Yaskawa INFORM job: aprem3TRJ2.JBI

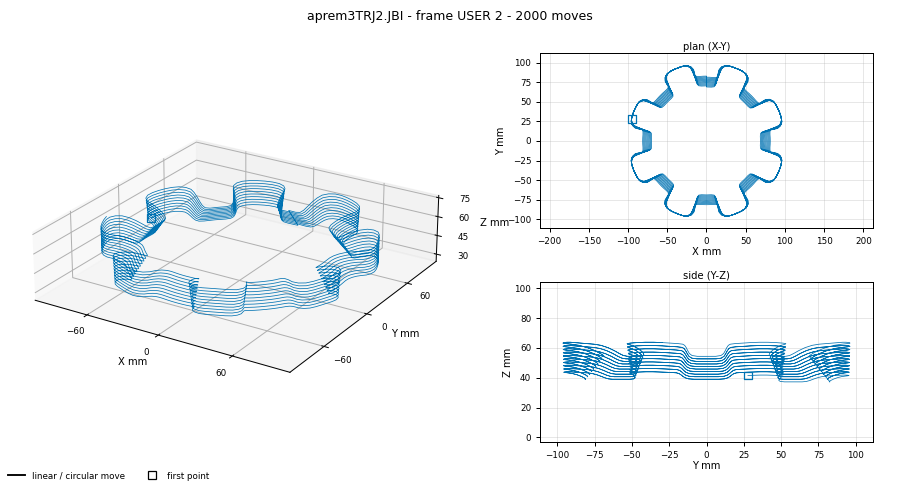
[picture p0: tool path of aprem3TRJ2.JBI in frame USER 2, 2000 of 2000 moves have a stored position in this frame; points joined in program order, loops and branches not executed]
/JOB
//NAME aprem3TRJ2
///FOLDERNAME DEMO
//POS
///NPOS 2000,0,2000,0,0,0
///USER 2
///TOOL 7
///POSTYPE USER
///RECTAN
///RCONF 1,0,0,0,0,0,0,0,0,0,0,0,0,0,0,0,0,0,0,0,0,0,0,0
C00000=-95.500,27.752,41.515,179.9573,-1.4576,-7126.2037
C00001=-94.679,31.992,41.678,179.9802,-0.0621,-7128.6701
C00002=-93.214,36.189,41.785,179.9968,-0.0083,-7131.2180
C00003=-91.502,40.323,41.785,179.9964,-0.0081,-7133.7821
C00004=-89.570,44.326,41.678,179.9701,-0.0579,-7136.3297
C00005=-87.153,47.905,41.515,178.9994,-1.0610,-7138.7961
C00006=-83.964,50.341,41.355,177.9940,-1.0426,-7140.9450
C00007=-80.606,51.270,41.159,176.0647,-0.0633,-7142.4587
C00008=-77.545,50.645,40.789,176.2827,1.1365,-7143.1487
C00009=-74.511,49.565,40.048,179.1830,0.2954,-7143.6320
C00010=-71.724,48.673,39.090,-174.7304,-1.4587,-7144.1614
C00011=-69.261,48.447,38.165,-161.9042,-0.3246,-7144.9722
C00012=-66.868,49.465,37.495,-150.0988,20.4873,-7146.4919
C00013=-64.059,52.288,37.229,-152.5931,29.6910,-7149.2230
C00014=-61.349,55.398,37.217,-152.6199,30.0136,-7152.0820
C00015=-58.451,58.451,37.225,-151.2604,28.7392,-7155.0000
C00016=-55.398,61.349,37.217,-149.9866,27.3805,-7157.9180
C00017=-52.288,64.059,37.229,-150.3100,27.4077,-7160.7770
C00018=-49.465,66.868,37.495,-159.5118,29.9009,-7163.5081
C00019=-48.447,69.261,38.165,179.6754,18.0958,-7165.0278
C00020=-48.673,71.724,39.090,178.5413,5.2696,-7165.8386
C00021=-49.565,74.511,40.048,-179.7046,-0.8170,-7166.3680
C00022=-50.645,77.545,40.789,-178.8635,-3.7173,-7166.8513
C00023=-51.270,80.606,41.159,179.9367,-3.9353,-7167.5413
C00024=-50.341,83.964,41.355,178.9574,-2.0060,-7169.0550
C00025=-47.905,87.153,41.515,178.9390,-1.0006,-7171.2039
C00026=-44.326,89.570,41.678,179.9421,-0.0299,-7173.6703
C00027=-40.323,91.502,41.785,179.9919,-0.0036,-7176.2179
C00028=-36.189,93.214,41.785,179.9917,-0.0032,-7178.7820
C00029=-31.992,94.679,41.678,179.9379,-0.0198,-7181.3299
C00030=-27.752,95.500,41.515,178.5424,-0.0427,-7183.7963
C00031=-23.775,94.968,41.355,177.8447,0.6817,-7185.9450
C00032=-20.743,93.250,41.159,177.1705,2.7402,-7187.4590
C00033=-19.021,90.644,40.789,178.1721,3.4318,-7188.1488
C00034=-17.640,87.735,40.048,179.6311,0.7865,-7188.6317
C00035=-16.299,85.134,39.090,-177.2970,-4.7574,-7189.1618
C00036=-14.718,83.232,38.165,-167.2077,-13.2282,-7189.9720
C00037=-12.305,82.260,37.495,-146.1451,-8.1050,-7191.4924
C00038=-8.324,82.270,37.229,-142.4105,2.0911,-7194.2225
C00039=-4.208,82.553,37.217,-142.2353,2.4190,-7197.0820
C00040=0.000,82.662,37.225,-142.2055,0.0004,-7200.0000
C00041=0.000,81.307,38.958,-141.7581,0.0003,-7200.0000
C00042=4.084,81.202,38.949,-141.7876,-2.4412,-7202.8792
C00043=8.115,80.931,38.962,-141.9747,-1.8578,-7205.7259
C00044=12.050,80.963,39.253,-146.2950,9.3084,-7208.4654
C00045=14.402,82.041,39.987,-169.0753,12.6711,-7209.9566
C00046=15.932,84.113,41.004,-178.0957,3.7141,-7210.7254
C00047=17.234,86.943,42.060,179.2930,-1.6621,-7211.2119
C00048=18.580,90.119,42.880,177.9599,-4.2630,-7211.6495
C00049=20.259,92.987,43.289,176.7690,-3.4884,-7212.2909
C00050=23.317,94.913,43.506,177.4450,-0.9091,-7213.8024
C00051=27.389,95.566,43.684,178.3657,0.0207,-7215.9922
C00052=31.762,94.755,43.864,179.9236,0.0242,-7218.5312
C00053=36.110,93.244,43.984,179.9901,0.0038,-7221.1696
C00054=40.400,91.468,43.984,179.9903,0.0044,-7223.8303
C00055=44.543,89.461,43.864,179.9289,0.0369,-7226.4689
C00056=48.209,86.942,43.684,178.8296,1.1411,-7229.0082
C00057=50.626,83.601,43.506,178.8351,2.4492,-7231.1977
C00058=51.426,80.077,43.289,-179.8173,4.7459,-7232.7089
C00059=50.586,76.861,42.880,-178.4237,4.4542,-7233.3509
C00060=49.291,73.664,42.060,-179.3244,1.6751,-7233.7878
C00061=48.211,70.742,41.004,178.7173,-3.9706,-7234.2746
C00062=47.828,68.195,39.987,178.7113,-16.4605,-7235.0436
C00063=48.729,65.770,39.253,-160.4159,-30.4372,-7236.5348
C00064=51.488,62.965,38.962,-150.0628,-27.9244,-7239.2737
C00065=54.531,60.307,38.949,-149.5942,-27.7685,-7242.1206
C00066=57.493,57.493,38.958,-150.8703,-29.1301,-7245.0000
C00067=60.306,54.531,38.949,-152.2311,-30.4055,-7247.8789
C00068=62.965,51.488,38.962,-152.0747,-29.9361,-7250.7263
C00069=65.770,48.729,39.253,-149.5629,-19.5850,-7253.4652
C00070=68.195,47.828,39.987,-163.5395,1.2887,-7254.9564
C00071=70.742,48.211,41.004,-176.0294,1.2827,-7255.7254
C00072=73.664,49.291,42.060,178.3249,-0.6756,-7256.2122
C00073=76.861,50.586,42.880,175.5458,-1.5763,-7256.6491
C00074=80.077,51.426,43.289,175.2541,-0.1827,-7257.2911
C00075=83.601,50.626,43.506,177.5508,1.1649,-7258.8023
C00076=86.942,48.209,43.684,178.8589,1.1704,-7260.9918
C00077=89.461,44.543,43.864,179.9631,0.0711,-7263.5311
C00078=91.468,40.400,43.984,179.9956,0.0097,-7266.1697
C00079=93.244,36.110,43.984,179.9962,0.0099,-7268.8304
C00080=94.755,31.762,43.864,179.9758,0.0764,-7271.4688
C00081=95.566,27.389,43.684,179.9793,1.6343,-7274.0078
C00082=94.913,23.317,43.506,-179.0909,2.5550,-7276.1976
C00083=92.987,20.259,43.289,-176.5116,3.2310,-7277.7091
C00084=90.119,18.580,42.880,-175.7370,2.0401,-7278.3505
C00085=86.943,17.234,42.060,-178.3379,0.7070,-7278.7881
C00086=84.113,15.932,41.004,176.2859,-1.9043,-7279.2746
C00087=82.041,14.402,39.987,167.3289,-10.9247,-7280.0434
C00088=80.963,12.050,39.253,170.6916,-33.7050,-7281.5346
C00089=80.931,8.115,38.962,-178.1422,-38.0253,-7284.2741
C00090=81.202,4.084,38.949,-177.5588,-38.2124,-7287.1208
C00091=81.307,0.000,38.958,179.9997,-38.2419,-7290.0000
C00092=81.202,-4.084,38.949,177.5593,-38.2124,-7292.8792
C00093=80.931,-8.116,38.962,178.1440,-38.0251,-7295.7266
C00094=80.963,-12.050,39.253,-170.6925,-33.7054,-7298.4654
C00095=82.041,-14.402,39.987,-167.3289,-10.9247,-7299.9566
C00096=84.113,-15.932,41.004,-176.2859,-1.9043,-7300.7254
C00097=86.943,-17.234,42.060,178.3379,0.7070,-7301.2119
C00098=90.119,-18.580,42.880,175.7370,2.0401,-7301.6495
C00099=92.987,-20.259,43.289,176.5116,3.2310,-7302.2909
C00100=94.913,-23.317,43.506,179.0909,2.5550,-7303.8024
C00101=95.566,-27.389,43.684,-179.9793,1.6343,-7305.9922
C00102=94.755,-31.762,43.864,-179.9758,0.0764,-7308.5312
C00103=93.244,-36.110,43.984,-179.9962,0.0099,-7311.1696
C00104=91.468,-40.400,43.984,-179.9956,0.0097,-7313.8303
C00105=89.461,-44.543,43.864,-179.9631,0.0711,-7316.4689
C00106=86.942,-48.209,43.684,-178.8589,1.1704,-7319.0082
C00107=83.601,-50.626,43.506,-177.5508,1.1649,-7321.1977
C00108=80.077,-51.426,43.289,-175.2541,-0.1827,-7322.7089
C00109=76.861,-50.586,42.880,-175.5458,-1.5763,-7323.3509
C00110=73.664,-49.291,42.060,-178.3249,-0.6756,-7323.7878
C00111=70.742,-48.211,41.004,176.0294,1.2827,-7324.2746
C00112=68.195,-47.828,39.987,163.5395,1.2887,-7325.0436
C00113=65.770,-48.729,39.253,149.5628,-19.5841,-7326.5348
C00114=62.965,-51.488,38.962,152.0756,-29.9372,-7329.2737
C00115=60.307,-54.531,38.949,152.2315,-30.4058,-7332.1206
C00116=57.493,-57.493,38.958,150.8699,-29.1297,-7335.0000
C00117=54.531,-60.306,38.949,149.5945,-27.7689,-7337.8789
C00118=51.488,-62.965,38.962,150.0639,-27.9253,-7340.7263
C00119=48.729,-65.770,39.253,160.4150,-30.4371,-7343.4652
C00120=47.828,-68.195,39.987,-178.7113,-16.4605,-7344.9564
C00121=48.211,-70.742,41.004,-178.7173,-3.9706,-7345.7254
C00122=49.291,-73.664,42.060,179.3244,1.6751,-7346.2122
C00123=50.586,-76.861,42.880,178.4237,4.4542,-7346.6491
C00124=51.426,-80.077,43.289,179.8173,4.7459,-7347.2911
C00125=50.626,-83.601,43.506,-178.8351,2.4492,-7348.8023
C00126=48.209,-86.942,43.684,-178.8296,1.1411,-7350.9918
C00127=44.543,-89.461,43.864,-179.9289,0.0369,-7353.5311
C00128=40.400,-91.468,43.984,-179.9903,0.0044,-7356.1697
C00129=36.110,-93.244,43.984,-179.9901,0.0038,-7358.8304
C00130=31.762,-94.755,43.864,-179.9236,0.0242,-7361.4688
C00131=27.389,-95.566,43.684,-178.3657,0.0207,-7364.0078
C00132=23.317,-94.913,43.506,-177.4450,-0.9091,-7366.1976
C00133=20.259,-92.987,43.289,-176.7690,-3.4884,-7367.7091
C00134=18.580,-90.119,42.880,-177.9599,-4.2630,-7368.3505
C00135=17.234,-86.943,42.060,-179.2930,-1.6621,-7368.7881
C00136=15.932,-84.113,41.004,178.0957,3.7141,-7369.2746
C00137=14.402,-82.041,39.987,169.0753,12.6711,-7370.0434
C00138=12.050,-80.963,39.253,146.2950,9.3084,-7371.5346
C00139=8.115,-80.931,38.962,141.9747,-1.8578,-7374.2741
C00140=4.084,-81.202,38.949,141.7876,-2.4412,-7377.1208
C00141=0.000,-81.307,38.958,141.7581,0.0003,-7380.0000
C00142=0.000,-81.307,38.958,141.7581,0.0003,-7380.0000
C00143=-4.084,-81.202,38.949,141.7876,2.4407,-7382.8792
C00144=-8.116,-80.931,38.962,141.9749,1.8560,-7385.7266
C00145=-12.050,-80.963,39.253,146.2946,-9.3075,-7388.4654
C00146=-14.402,-82.041,39.987,169.0753,-12.6711,-7389.9566
C00147=-15.932,-84.113,41.004,178.0957,-3.7141,-7390.7254
C00148=-17.234,-86.943,42.060,-179.2930,1.6621,-7391.2119
C00149=-18.580,-90.119,42.880,-177.9599,4.2630,-7391.6495
C00150=-20.259,-92.987,43.289,-176.7690,3.4884,-7392.2909
C00151=-23.317,-94.913,43.506,-177.4450,0.9091,-7393.8024
C00152=-27.389,-95.566,43.684,-178.3657,-0.0207,-7395.9922
C00153=-31.762,-94.755,43.864,-179.9236,-0.0242,-7398.5312
C00154=-36.110,-93.244,43.984,-179.9901,-0.0038,-7401.1696
C00155=-40.400,-91.468,43.984,-179.9903,-0.0044,-7403.8303
C00156=-44.543,-89.461,43.864,-179.9289,-0.0369,-7406.4689
C00157=-48.209,-86.942,43.684,-178.8296,-1.1411,-7409.0082
C00158=-50.626,-83.601,43.506,-178.8351,-2.4492,-7411.1977
C00159=-51.426,-80.077,43.289,179.8173,-4.7459,-7412.7089
C00160=-50.586,-76.861,42.880,178.4237,-4.4542,-7413.3509
C00161=-49.291,-73.664,42.060,179.3244,-1.6751,-7413.7878
C00162=-48.211,-70.742,41.004,-178.7173,3.9706,-7414.2746
C00163=-47.828,-68.195,39.987,-178.7113,16.4605,-7415.0436
C00164=-48.729,-65.770,39.253,160.4159,30.4372,-7416.5348
C00165=-51.488,-62.965,38.962,150.0628,27.9244,-7419.2737
C00166=-54.531,-60.307,38.949,149.5942,27.7685,-7422.1206
C00167=-57.493,-57.493,38.958,150.8703,29.1301,-7425.0000
C00168=-60.306,-54.531,38.949,152.2311,30.4055,-7427.8789
C00169=-62.965,-51.488,38.962,152.0747,29.9361,-7430.7263
C00170=-65.770,-48.729,39.253,149.5629,19.5850,-7433.4652
C00171=-68.195,-47.828,39.987,163.5395,-1.2887,-7434.9564
C00172=-70.742,-48.211,41.004,176.0294,-1.2827,-7435.7254
C00173=-73.664,-49.291,42.060,-178.3249,0.6756,-7436.2122
C00174=-76.861,-50.586,42.880,-175.5458,1.5763,-7436.6491
C00175=-80.077,-51.426,43.289,-175.2541,0.1827,-7437.2911
C00176=-83.601,-50.626,43.506,-177.5508,-1.1649,-7438.8023
C00177=-86.942,-48.209,43.684,-178.8589,-1.1704,-7440.9918
C00178=-89.461,-44.543,43.864,-179.9631,-0.0711,-7443.5311
C00179=-91.468,-40.400,43.984,-179.9956,-0.0097,-7446.1697
C00180=-93.244,-36.110,43.984,-179.9962,-0.0099,-7448.8304
C00181=-94.755,-31.762,43.864,-179.9758,-0.0764,-7451.4688
C00182=-95.566,-27.389,43.684,-179.9793,-1.6343,-7454.0078
C00183=-94.913,-23.317,43.506,179.0909,-2.5550,-7456.1976
C00184=-92.987,-20.259,43.289,176.5116,-3.2310,-7457.7091
C00185=-90.119,-18.580,42.880,175.7370,-2.0401,-7458.3505
C00186=-86.943,-17.234,42.060,178.3379,-0.7070,-7458.7881
C00187=-84.113,-15.932,41.004,-176.2859,1.9043,-7459.2746
C00188=-82.041,-14.402,39.987,-167.3289,10.9247,-7460.0434
C00189=-80.963,-12.050,39.253,-170.6916,33.7050,-7461.5346
C00190=-80.931,-8.115,38.962,178.1422,38.0253,-7464.2741
C00191=-81.202,-4.084,38.949,177.5588,38.2124,-7467.1208
C00192=-81.307,0.000,38.958,-179.9997,38.2419,-7470.0000
C00193=-81.202,4.084,38.949,-177.5593,38.2124,-7472.8792
C00194=-80.931,8.116,38.962,-178.1440,38.0251,-7475.7266
C00195=-80.963,12.050,39.253,170.6925,33.7054,-7478.4654
C00196=-82.041,14.402,39.987,167.3289,10.9247,-7479.9566
C00197=-84.113,15.932,41.004,176.2859,1.9043,-7480.7254
C00198=-86.943,17.234,42.060,-178.3379,-0.7070,-7481.2119
C00199=-90.119,18.580,42.880,-175.7370,-2.0401,-7481.6495
C00200=-92.987,20.259,43.289,-176.5116,-3.2310,-7482.2909
C00201=-94.913,23.317,43.506,-179.0909,-2.5550,-7483.8024
C00202=-95.566,27.389,43.684,179.9793,-1.6343,-7485.9922
C00203=-94.755,31.762,43.864,179.9758,-0.0764,-7488.5312
C00204=-93.244,36.110,43.984,179.9962,-0.0099,-7491.1696
C00205=-91.468,40.400,43.984,179.9956,-0.0097,-7493.8303
C00206=-89.461,44.543,43.864,179.9631,-0.0711,-7496.4689
C00207=-86.942,48.209,43.684,178.8589,-1.1704,-7499.0082
C00208=-83.601,50.626,43.506,177.5508,-1.1649,-7501.1977
C00209=-80.077,51.426,43.289,175.2541,0.1827,-7502.7089
C00210=-76.861,50.586,42.880,175.5458,1.5763,-7503.3509
C00211=-73.664,49.291,42.060,178.3249,0.6756,-7503.7878
C00212=-70.742,48.211,41.004,-176.0294,-1.2827,-7504.2746
C00213=-68.195,47.828,39.987,-163.5395,-1.2887,-7505.0436
C00214=-65.770,48.729,39.253,-149.5628,19.5841,-7506.5348
C00215=-62.965,51.488,38.962,-152.0756,29.9372,-7509.2737
C00216=-60.307,54.531,38.949,-152.2315,30.4058,-7512.1206
C00217=-57.493,57.493,38.958,-150.8699,29.1297,-7515.0000
C00218=-54.531,60.306,38.949,-149.5945,27.7689,-7517.8789
C00219=-51.488,62.965,38.962,-150.0639,27.9253,-7520.7263
C00220=-48.729,65.770,39.253,-160.4150,30.4371,-7523.4652
C00221=-47.828,68.195,39.987,178.7113,16.4605,-7524.9564
C00222=-48.211,70.742,41.004,178.7173,3.9706,-7525.7254
C00223=-49.291,73.664,42.060,-179.3244,-1.6751,-7526.2122
C00224=-50.586,76.861,42.880,-178.4237,-4.4542,-7526.6491
C00225=-51.426,80.077,43.289,-179.8173,-4.7459,-7527.2911
C00226=-50.626,83.601,43.506,178.8351,-2.4492,-7528.8023
C00227=-48.209,86.942,43.684,178.8296,-1.1411,-7530.9918
C00228=-44.543,89.461,43.864,179.9289,-0.0369,-7533.5311
C00229=-40.400,91.468,43.984,179.9903,-0.0044,-7536.1697
C00230=-36.110,93.244,43.984,179.9901,-0.0038,-7538.8304
C00231=-31.762,94.755,43.864,179.9236,-0.0242,-7541.4688
C00232=-27.389,95.566,43.684,178.3657,-0.0207,-7544.0078
C00233=-23.317,94.913,43.506,177.4450,0.9091,-7546.1976
C00234=-20.259,92.987,43.289,176.7690,3.4884,-7547.7091
C00235=-18.580,90.119,42.880,177.9599,4.2630,-7548.3505
C00236=-17.234,86.943,42.060,179.2930,1.6621,-7548.7881
C00237=-15.932,84.113,41.004,-178.0957,-3.7141,-7549.2746
C00238=-14.402,82.041,39.987,-169.0753,-12.6711,-7550.0434
C00239=-12.050,80.963,39.253,-146.2946,-9.3075,-7551.5346
C00240=-8.116,80.931,38.962,-141.9749,1.8560,-7554.2734
C00241=-4.084,81.202,38.949,-141.7876,2.4407,-7557.1208
C00242=0.000,81.307,38.958,-141.7581,0.0003,-7560.0000
C00243=0.000,79.940,40.681,-141.3945,0.0003,-7560.0000
C00244=3.959,79.840,40.672,-141.4236,-2.4543,-7562.8388
C00245=7.905,79.580,40.686,-141.6255,-1.5989,-7565.6728
C00246=11.791,79.654,41.003,-146.5959,10.4668,-7568.4202
C00247=14.083,80.839,41.802,-170.8088,11.8957,-7569.8823
C00248=15.561,83.082,42.912,-178.7432,2.6994,-7570.6084
C00249=16.825,86.143,44.068,179.0449,-2.4598,-7571.0516
C00250=18.134,89.588,44.968,177.8329,-5.0059,-7571.4429
C00251=19.771,92.721,45.418,176.4774,-4.2024,-7572.0370
C00252=22.856,94.857,45.657,177.0847,-1.1491,-7573.5473
C00253=27.022,95.633,45.852,178.2015,-0.0057,-7575.7781
C00254=31.529,94.831,46.051,179.9101,0.0282,-7578.3907
C00255=36.031,93.275,46.182,179.9885,0.0043,-7581.1209
C00256=40.478,91.433,46.182,179.9888,0.0050,-7583.8793
C00257=44.762,89.350,46.051,179.9165,0.0436,-7586.6097
C00258=48.515,86.730,45.852,178.7321,1.2760,-7589.2218
C00259=50.913,83.236,45.657,178.7496,2.8735,-7591.4529
C00260=51.583,79.544,45.418,-179.5172,5.4544,-7592.9628
C00261=50.526,76.172,44.968,-177.9852,5.0686,-7593.5569
C00262=49.015,72.810,44.068,-178.9351,2.4144,-7593.9481
C00263=47.744,69.752,42.912,178.9787,-2.7968,-7594.3909
C00264=47.203,67.120,41.802,178.0217,-14.7549,-7595.1173
C00265=47.986,64.662,41.003,-161.4435,-30.8352,-7596.5793
C00266=50.682,61.862,40.686,-149.9004,-28.3778,-7599.3269
C00267=53.655,59.255,40.672,-149.2767,-28.0885,-7602.1606
C00268=56.526,56.526,40.681,-150.5516,-29.4487,-7605.0000
C00269=59.255,53.656,40.672,-151.9113,-30.7231,-7607.8388
C00270=61.862,50.682,40.686,-151.6213,-30.0984,-7610.6731
C00271=64.662,47.986,41.003,-149.1649,-18.5575,-7613.4207
C00272=67.120,47.203,41.802,-165.2451,1.9783,-7614.8827
C00273=69.752,47.744,42.912,-177.2032,1.0213,-7615.6091
C00274=72.810,49.015,44.068,177.5856,-1.0649,-7616.0519
C00275=76.172,50.526,44.968,174.9314,-2.0148,-7616.4431
C00276=79.544,51.583,45.418,174.5456,-0.4828,-7617.0372
C00277=83.236,50.913,45.657,177.1265,1.2504,-7618.5471
C00278=86.730,48.515,45.852,178.7240,1.2679,-7620.7782
C00279=89.350,44.762,46.051,179.9564,0.0835,-7623.3903
C00280=91.433,40.478,46.182,179.9950,0.0112,-7626.1207
C00281=93.275,36.031,46.182,179.9957,0.0115,-7628.8791
C00282=94.831,31.529,46.051,179.9718,0.0899,-7631.6093
C00283=95.633,27.022,45.852,-179.9943,1.7985,-7634.2219
C00284=94.857,22.856,45.657,-178.8509,2.9153,-7636.4527
C00285=92.721,19.771,45.418,-175.7976,3.5226,-7637.9630
C00286=89.588,18.134,44.968,-174.9941,2.1671,-7638.5571
C00287=86.143,16.825,44.068,-177.5402,0.9551,-7638.9484
C00288=83.082,15.561,42.912,177.3006,-1.2568,-7639.3916
C00289=80.839,14.083,41.802,168.1043,-9.1912,-7640.1177
C00290=79.654,11.791,41.003,169.5332,-33.4041,-7641.5798
C00291=79.580,7.905,40.686,-178.4011,-38.3745,-7644.3272
C00292=79.840,3.959,40.672,-177.5457,-38.5764,-7647.1612
C00293=79.940,0.000,40.681,179.9997,-38.6055,-7650.0000
C00294=79.840,-3.959,40.672,177.5462,-38.5764,-7652.8388
C00295=79.580,-7.905,40.686,178.4031,-38.3743,-7655.6728
C00296=79.654,-11.792,41.003,-169.5340,-33.4045,-7658.4209
C00297=80.839,-14.083,41.802,-168.1043,-9.1912,-7659.8823
C00298=83.082,-15.561,42.912,-177.3006,-1.2568,-7660.6084
C00299=86.143,-16.825,44.068,177.5402,0.9551,-7661.0516
C00300=89.588,-18.134,44.968,174.9941,2.1671,-7661.4429
C00301=92.721,-19.771,45.418,175.7976,3.5226,-7662.0370
C00302=94.857,-22.856,45.657,178.8509,2.9153,-7663.5473
C00303=95.633,-27.022,45.852,179.9943,1.7985,-7665.7781
C00304=94.831,-31.529,46.051,-179.9718,0.0899,-7668.3907
C00305=93.275,-36.031,46.182,-179.9957,0.0115,-7671.1209
C00306=91.433,-40.478,46.182,-179.9950,0.0112,-7673.8793
C00307=89.350,-44.762,46.051,-179.9564,0.0835,-7676.6097
C00308=86.730,-48.515,45.852,-178.7240,1.2679,-7679.2218
C00309=83.236,-50.913,45.657,-177.1265,1.2504,-7681.4529
C00310=79.544,-51.583,45.418,-174.5456,-0.4828,-7682.9628
C00311=76.172,-50.526,44.968,-174.9314,-2.0148,-7683.5569
C00312=72.810,-49.015,44.068,-177.5856,-1.0649,-7683.9481
C00313=69.752,-47.744,42.912,177.2032,1.0213,-7684.3909
C00314=67.120,-47.203,41.802,165.2451,1.9783,-7685.1173
C00315=64.662,-47.986,41.003,149.1648,-18.5565,-7686.5793
C00316=61.862,-50.682,40.686,151.6222,-30.0996,-7689.3269
C00317=59.255,-53.655,40.672,151.9115,-30.7233,-7692.1606
C00318=56.526,-56.526,40.681,150.5513,-29.4484,-7695.0000
C00319=53.656,-59.255,40.672,149.2769,-28.0887,-7697.8388
C00320=50.682,-61.862,40.686,149.9016,-28.3787,-7700.6731
C00321=47.986,-64.662,41.003,161.4425,-30.8351,-7703.4207
C00322=47.203,-67.120,41.802,-178.0217,-14.7549,-7704.8827
C00323=47.744,-69.752,42.912,-178.9787,-2.7968,-7705.6091
C00324=49.015,-72.810,44.068,178.9351,2.4144,-7706.0519
C00325=50.526,-76.172,44.968,177.9852,5.0686,-7706.4431
C00326=51.583,-79.544,45.418,179.5172,5.4544,-7707.0372
C00327=50.913,-83.236,45.657,-178.7496,2.8735,-7708.5471
C00328=48.515,-86.730,45.852,-178.7321,1.2760,-7710.7782
C00329=44.762,-89.350,46.051,-179.9165,0.0436,-7713.3903
C00330=40.478,-91.433,46.182,-179.9888,0.0050,-7716.1207
C00331=36.031,-93.275,46.182,-179.9885,0.0043,-7718.8791
C00332=31.529,-94.831,46.051,-179.9101,0.0282,-7721.6093
C00333=27.022,-95.633,45.852,-178.2015,-0.0057,-7724.2219
C00334=22.856,-94.857,45.657,-177.0847,-1.1491,-7726.4527
C00335=19.771,-92.721,45.418,-176.4774,-4.2024,-7727.9630
C00336=18.134,-89.588,44.968,-177.8329,-5.0059,-7728.5571
C00337=16.825,-86.143,44.068,-179.0449,-2.4598,-7728.9484
C00338=15.561,-83.082,42.912,178.7432,2.6994,-7729.3916
C00339=14.083,-80.839,41.802,170.8088,11.8957,-7730.1177
C00340=11.791,-79.654,41.003,146.5959,10.4668,-7731.5798
C00341=7.905,-79.580,40.686,141.6255,-1.5989,-7734.3272
C00342=3.959,-79.840,40.672,141.4236,-2.4543,-7737.1612
C00343=0.000,-79.940,40.681,141.3945,0.0003,-7740.0000
C00344=0.000,-79.940,40.681,141.3945,0.0003,-7740.0000
C00345=-3.959,-79.840,40.672,141.4236,2.4538,-7742.8388
C00346=-7.905,-79.580,40.686,141.6257,1.5969,-7745.6728
C00347=-11.792,-79.654,41.003,146.5955,-10.4660,-7748.4209
C00348=-14.083,-80.839,41.802,170.8088,-11.8957,-7749.8823
C00349=-15.561,-83.082,42.912,178.7432,-2.6994,-7750.6084
C00350=-16.825,-86.143,44.068,-179.0449,2.4598,-7751.0516
C00351=-18.134,-89.588,44.968,-177.8329,5.0059,-7751.4429
C00352=-19.771,-92.721,45.418,-176.4774,4.2024,-7752.0370
C00353=-22.856,-94.857,45.657,-177.0847,1.1491,-7753.5473
C00354=-27.022,-95.633,45.852,-178.2015,0.0057,-7755.7781
C00355=-31.529,-94.831,46.051,-179.9101,-0.0282,-7758.3907
C00356=-36.031,-93.275,46.182,-179.9885,-0.0043,-7761.1209
C00357=-40.478,-91.433,46.182,-179.9888,-0.0050,-7763.8793
C00358=-44.762,-89.350,46.051,-179.9165,-0.0436,-7766.6097
C00359=-48.515,-86.730,45.852,-178.7321,-1.2760,-7769.2218
C00360=-50.913,-83.236,45.657,-178.7496,-2.8735,-7771.4529
C00361=-51.583,-79.544,45.418,179.5172,-5.4544,-7772.9628
C00362=-50.526,-76.172,44.968,177.9852,-5.0686,-7773.5569
C00363=-49.015,-72.810,44.068,178.9351,-2.4144,-7773.9481
C00364=-47.744,-69.752,42.912,-178.9787,2.7968,-7774.3909
C00365=-47.203,-67.120,41.802,-178.0217,14.7549,-7775.1173
C00366=-47.986,-64.662,41.003,161.4435,30.8352,-7776.5793
C00367=-50.682,-61.862,40.686,149.9004,28.3778,-7779.3269
C00368=-53.655,-59.255,40.672,149.2767,28.0885,-7782.1606
C00369=-56.526,-56.526,40.681,150.5516,29.4487,-7785.0000
C00370=-59.255,-53.656,40.672,151.9113,30.7231,-7787.8388
C00371=-61.862,-50.682,40.686,151.6213,30.0984,-7790.6731
C00372=-64.662,-47.986,41.003,149.1649,18.5575,-7793.4207
C00373=-67.120,-47.203,41.802,165.2451,-1.9783,-7794.8827
C00374=-69.752,-47.744,42.912,177.2032,-1.0213,-7795.6091
C00375=-72.810,-49.015,44.068,-177.5856,1.0649,-7796.0519
C00376=-76.172,-50.526,44.968,-174.9314,2.0148,-7796.4431
C00377=-79.544,-51.583,45.418,-174.5456,0.4828,-7797.0372
C00378=-83.236,-50.913,45.657,-177.1265,-1.2504,-7798.5471
C00379=-86.730,-48.515,45.852,-178.7240,-1.2679,-7800.7782
C00380=-89.350,-44.762,46.051,-179.9564,-0.0835,-7803.3903
C00381=-91.433,-40.478,46.182,-179.9950,-0.0112,-7806.1207
C00382=-93.275,-36.031,46.182,-179.9957,-0.0115,-7808.8791
C00383=-94.831,-31.529,46.051,-179.9718,-0.0899,-7811.6093
C00384=-95.633,-27.022,45.852,179.9943,-1.7985,-7814.2219
C00385=-94.857,-22.856,45.657,178.8509,-2.9153,-7816.4527
C00386=-92.721,-19.771,45.418,175.7976,-3.5226,-7817.9630
C00387=-89.588,-18.134,44.968,174.9941,-2.1671,-7818.5571
C00388=-86.143,-16.825,44.068,177.5402,-0.9551,-7818.9484
C00389=-83.082,-15.561,42.912,-177.3006,1.2568,-7819.3916
C00390=-80.839,-14.083,41.802,-168.1043,9.1912,-7820.1177
C00391=-79.654,-11.791,41.003,-169.5332,33.4041,-7821.5798
C00392=-79.580,-7.905,40.686,178.4011,38.3745,-7824.3272
C00393=-79.840,-3.959,40.672,177.5457,38.5764,-7827.1612
C00394=-79.940,0.000,40.681,-179.9997,38.6055,-7830.0000
C00395=-79.840,3.959,40.672,-177.5462,38.5764,-7832.8388
C00396=-79.580,7.905,40.686,-178.4031,38.3743,-7835.6728
C00397=-79.654,11.792,41.003,169.5340,33.4045,-7838.4209
C00398=-80.839,14.083,41.802,168.1043,9.1912,-7839.8823
C00399=-83.082,15.561,42.912,177.3006,1.2568,-7840.6084
C00400=-86.143,16.825,44.068,-177.5402,-0.9551,-7841.0516
C00401=-89.588,18.134,44.968,-174.9941,-2.1671,-7841.4429
C00402=-92.721,19.771,45.418,-175.7976,-3.5226,-7842.0370
C00403=-94.857,22.856,45.657,-178.8509,-2.9153,-7843.5473
C00404=-95.633,27.022,45.852,-179.9943,-1.7985,-7845.7781
C00405=-94.831,31.529,46.051,179.9718,-0.0899,-7848.3907
C00406=-93.275,36.031,46.182,179.9957,-0.0115,-7851.1209
C00407=-91.433,40.478,46.182,179.9950,-0.0112,-7853.8793
C00408=-89.350,44.762,46.051,179.9564,-0.0835,-7856.6097
C00409=-86.730,48.515,45.852,178.7240,-1.2679,-7859.2218
C00410=-83.236,50.913,45.657,177.1265,-1.2504,-7861.4529
C00411=-79.544,51.583,45.418,174.5456,0.4828,-7862.9628
C00412=-76.172,50.526,44.968,174.9314,2.0148,-7863.5569
C00413=-72.810,49.015,44.068,177.5856,1.0649,-7863.9481
C00414=-69.752,47.744,42.912,-177.2032,-1.0213,-7864.3909
C00415=-67.120,47.203,41.802,-165.2451,-1.9783,-7865.1173
C00416=-64.662,47.986,41.003,-149.1648,18.5565,-7866.5793
C00417=-61.862,50.682,40.686,-151.6222,30.0996,-7869.3269
C00418=-59.255,53.655,40.672,-151.9115,30.7233,-7872.1606
C00419=-56.526,56.526,40.681,-150.5513,29.4484,-7875.0000
C00420=-53.656,59.255,40.672,-149.2769,28.0887,-7877.8388
C00421=-50.682,61.862,40.686,-149.9016,28.3787,-7880.6731
C00422=-47.986,64.662,41.003,-161.4425,30.8351,-7883.4207
C00423=-47.203,67.120,41.802,178.0217,14.7549,-7884.8827
C00424=-47.744,69.752,42.912,178.9787,2.7968,-7885.6091
C00425=-49.015,72.810,44.068,-178.9351,-2.4144,-7886.0519
C00426=-50.526,76.172,44.968,-177.9852,-5.0686,-7886.4431
C00427=-51.583,79.544,45.418,-179.5172,-5.4544,-7887.0372
C00428=-50.913,83.236,45.657,178.7496,-2.8735,-7888.5471
C00429=-48.515,86.730,45.852,178.7321,-1.2760,-7890.7782
C00430=-44.762,89.350,46.051,179.9165,-0.0436,-7893.3903
C00431=-40.478,91.433,46.182,179.9888,-0.0050,-7896.1207
C00432=-36.031,93.275,46.182,179.9885,-0.0043,-7898.8791
C00433=-31.529,94.831,46.051,179.9101,-0.0282,-7901.6093
C00434=-27.022,95.633,45.852,178.2015,0.0057,-7904.2219
C00435=-22.856,94.857,45.657,177.0847,1.1491,-7906.4527
C00436=-19.771,92.721,45.418,176.4774,4.2024,-7907.9630
C00437=-18.134,89.588,44.968,177.8329,5.0059,-7908.5571
C00438=-16.825,86.143,44.068,179.0449,2.4598,-7908.9484
C00439=-15.561,83.082,42.912,-178.7432,-2.6994,-7909.3916
C00440=-14.083,80.839,41.802,-170.8088,-11.8957,-7910.1177
C00441=-11.792,79.654,41.003,-146.5955,-10.4660,-7911.5791
C00442=-7.905,79.580,40.686,-141.6257,1.5969,-7914.3272
C00443=-3.959,79.840,40.672,-141.4236,2.4538,-7917.1612
C00444=0.000,79.940,40.681,-141.3945,0.0003,-7920.0000
C00445=0.000,78.562,42.397,-141.1109,0.0002,-7920.0000
C00446=3.833,78.467,42.387,-141.1396,-2.4588,-7922.7966
C00447=7.694,78.220,42.402,-141.3590,-1.3181,-7925.6177
C00448=11.532,78.336,42.745,-147.0431,11.5605,-7928.3745
C00449=13.762,79.628,43.611,-172.3770,10.9592,-7929.8055
C00450=15.189,82.045,44.816,-179.2626,1.7346,-7930.4884
C00451=16.414,85.339,46.074,178.8680,-3.1755,-7930.8872
C00452=17.687,89.056,47.055,177.7717,-5.6565,-7931.2331
C00453=19.281,92.454,47.546,176.2826,-4.8619,-7931.7800
C00454=22.392,94.802,47.807,176.7679,-1.3940,-7933.2896
C00455=26.654,95.700,48.020,178.0518,-0.0356,-7935.5634
C00456=31.296,94.909,48.237,179.8977,0.0319,-7938.2498
C00457=35.952,93.306,48.381,179.9872,0.0049,-7941.0723
C00458=40.555,91.399,48.381,179.9875,0.0056,-7943.9275
C00459=44.981,89.240,48.237,179.9051,0.0498,-7946.7502
C00460=48.823,86.517,48.020,178.6473,1.4030,-7949.4368
C00461=51.201,82.869,47.807,178.6983,3.2702,-7951.7100
C00462=51.741,79.009,47.546,-179.1862,6.0558,-7953.2198
C00463=50.465,75.478,47.055,-177.5651,5.5716,-7953.7669
C00464=48.737,71.950,46.074,-178.5531,3.0453,-7954.1127
C00465=47.275,68.755,44.816,179.2946,-1.7479,-7954.5119
C00466=46.575,66.037,43.611,177.5785,-13.0378,-7955.1948
C00467=47.238,63.546,42.745,-162.5779,-31.0935,-7956.6259
C00468=49.870,60.750,42.402,-149.8188,-28.7683,-7959.3828
C00469=52.774,58.195,42.387,-149.0312,-28.3421,-7962.2032
C00470=55.552,55.552,42.397,-150.3022,-29.6980,-7965.0000
C00471=58.195,52.774,42.387,-151.6576,-30.9686,-7967.7968
C00472=60.750,49.870,42.402,-151.2308,-30.1799,-7970.6172
C00473=63.546,47.238,42.745,-148.9065,-17.4230,-7973.3741
C00474=66.037,46.575,43.611,-166.9622,2.4215,-7974.8052
C00475=68.755,47.275,44.816,-178.2521,0.7054,-7975.4881
C00476=71.950,48.737,46.074,176.9547,-1.4469,-7975.8873
C00477=75.478,50.465,47.055,174.4284,-2.4349,-7976.2331
C00478=79.009,51.741,47.546,173.9442,-0.8138,-7976.7802
C00479=82.869,51.201,47.807,176.7298,1.3017,-7978.2900
C00480=86.517,48.823,48.020,178.5970,1.3527,-7980.5632
C00481=89.240,44.981,48.237,179.9502,0.0949,-7983.2498
C00482=91.399,40.555,48.381,179.9944,0.0125,-7986.0725
C00483=93.306,35.952,48.381,179.9951,0.0128,-7988.9277
C00484=94.909,31.296,48.237,179.9681,0.1023,-7991.7502
C00485=95.700,26.654,48.020,-179.9644,1.9482,-7994.4366
C00486=94.802,22.392,47.807,-178.6060,3.2321,-7996.7104
C00487=92.454,19.281,47.546,-175.1381,3.7174,-7998.2200
C00488=89.056,17.687,47.055,-174.3435,2.2283,-7998.7669
C00489=85.339,16.414,46.074,-176.8245,1.1320,-7999.1128
C00490=82.045,15.189,44.816,178.2654,-0.7374,-7999.5116
C00491=79.628,13.762,43.611,169.0408,-7.6230,-8000.1945
C00492=78.336,11.532,42.745,168.4395,-32.9569,-8001.6255
C00493=78.220,7.694,42.402,-178.6819,-38.6410,-8004.3823
C00494=78.467,3.833,42.387,-177.5412,-38.8604,-8007.2034
C00495=78.562,0.000,42.397,179.9998,-38.8891,-8010.0000
C00496=78.467,-3.833,42.387,177.5416,-38.8604,-8012.7966
C00497=78.220,-7.694,42.402,178.6839,-38.6407,-8015.6177
C00498=78.336,-11.532,42.745,-168.4403,-32.9573,-8018.3745
C00499=79.628,-13.762,43.611,-169.0408,-7.6230,-8019.8055
C00500=82.045,-15.189,44.816,-178.2654,-0.7374,-8020.4884
C00501=85.339,-16.414,46.074,176.8245,1.1320,-8020.8872
C00502=89.056,-17.687,47.055,174.3435,2.2283,-8021.2331
C00503=92.454,-19.281,47.546,175.1381,3.7174,-8021.7800
C00504=94.802,-22.392,47.807,178.6060,3.2321,-8023.2896
C00505=95.700,-26.654,48.020,179.9644,1.9482,-8025.5634
C00506=94.909,-31.296,48.237,-179.9681,0.1023,-8028.2498
C00507=93.306,-35.952,48.381,-179.9951,0.0128,-8031.0723
C00508=91.399,-40.555,48.381,-179.9944,0.0125,-8033.9275
C00509=89.240,-44.981,48.237,-179.9502,0.0949,-8036.7502
C00510=86.517,-48.823,48.020,-178.5970,1.3527,-8039.4368
C00511=82.869,-51.201,47.807,-176.7298,1.3017,-8041.7100
C00512=79.009,-51.741,47.546,-173.9442,-0.8138,-8043.2198
C00513=75.478,-50.465,47.055,-174.4284,-2.4349,-8043.7669
C00514=71.950,-48.737,46.074,-176.9547,-1.4469,-8044.1127
C00515=68.755,-47.275,44.816,178.2521,0.7054,-8044.5119
C00516=66.037,-46.575,43.611,166.9622,2.4215,-8045.1948
C00517=63.546,-47.238,42.745,148.9065,-17.4221,-8046.6259
C00518=60.750,-49.870,42.402,151.2317,-30.1812,-8049.3828
C00519=58.195,-52.774,42.387,151.6579,-30.9688,-8052.2032
C00520=55.552,-55.552,42.397,150.3020,-29.6978,-8055.0000
C00521=52.774,-58.195,42.387,149.0314,-28.3424,-8057.7968
C00522=49.870,-60.750,42.402,149.8201,-28.7692,-8060.6172
C00523=47.238,-63.546,42.745,162.5770,-31.0935,-8063.3741
C00524=46.575,-66.037,43.611,-177.5785,-13.0378,-8064.8052
C00525=47.275,-68.755,44.816,-179.2946,-1.7479,-8065.4881
C00526=48.737,-71.950,46.074,178.5531,3.0453,-8065.8873
C00527=50.465,-75.478,47.055,177.5651,5.5716,-8066.2331
C00528=51.741,-79.009,47.546,179.1862,6.0558,-8066.7802
C00529=51.201,-82.869,47.807,-178.6983,3.2702,-8068.2900
C00530=48.823,-86.517,48.020,-178.6473,1.4030,-8070.5632
C00531=44.981,-89.240,48.237,-179.9051,0.0498,-8073.2498
C00532=40.555,-91.399,48.381,-179.9875,0.0056,-8076.0725
C00533=35.952,-93.306,48.381,-179.9872,0.0049,-8078.9277
C00534=31.296,-94.909,48.237,-179.8977,0.0319,-8081.7502
C00535=26.654,-95.700,48.020,-178.0518,-0.0356,-8084.4366
C00536=22.392,-94.802,47.807,-176.7679,-1.3940,-8086.7104
C00537=19.281,-92.454,47.546,-176.2826,-4.8619,-8088.2200
C00538=17.687,-89.056,47.055,-177.7717,-5.6565,-8088.7669
C00539=16.414,-85.339,46.074,-178.8680,-3.1755,-8089.1128
C00540=15.189,-82.045,44.816,179.2626,1.7346,-8089.5116
C00541=13.762,-79.628,43.611,172.3770,10.9592,-8090.1945
C00542=11.532,-78.336,42.745,147.0431,11.5605,-8091.6255
C00543=7.694,-78.220,42.402,141.3590,-1.3181,-8094.3823
C00544=3.833,-78.467,42.387,141.1396,-2.4588,-8097.2034
C00545=0.000,-78.562,42.397,141.1109,0.0002,-8100.0000
C00546=0.000,-78.562,42.397,141.1109,0.0002,-8100.0000
C00547=-3.833,-78.467,42.387,141.1396,2.4584,-8102.7966
C00548=-7.694,-78.220,42.402,141.3593,1.3161,-8105.6177
C00549=-11.532,-78.336,42.745,147.0427,-11.5597,-8108.3745
C00550=-13.762,-79.628,43.611,172.3770,-10.9592,-8109.8055
C00551=-15.189,-82.045,44.816,179.2626,-1.7346,-8110.4884
C00552=-16.414,-85.339,46.074,-178.8680,3.1755,-8110.8872
C00553=-17.687,-89.056,47.055,-177.7717,5.6565,-8111.2331
C00554=-19.281,-92.454,47.546,-176.2826,4.8619,-8111.7800
C00555=-22.392,-94.802,47.807,-176.7679,1.3940,-8113.2896
C00556=-26.654,-95.700,48.020,-178.0518,0.0356,-8115.5634
C00557=-31.296,-94.909,48.237,-179.8977,-0.0319,-8118.2498
C00558=-35.952,-93.306,48.381,-179.9872,-0.0049,-8121.0723
C00559=-40.555,-91.399,48.381,-179.9875,-0.0056,-8123.9275
C00560=-44.981,-89.240,48.237,-179.9051,-0.0498,-8126.7502
C00561=-48.823,-86.517,48.020,-178.6473,-1.4030,-8129.4368
C00562=-51.201,-82.869,47.807,-178.6983,-3.2702,-8131.7100
C00563=-51.741,-79.009,47.546,179.1862,-6.0558,-8133.2198
C00564=-50.465,-75.478,47.055,177.5651,-5.5716,-8133.7669
C00565=-48.737,-71.950,46.074,178.5531,-3.0453,-8134.1127
C00566=-47.275,-68.755,44.816,-179.2946,1.7479,-8134.5119
C00567=-46.575,-66.037,43.611,-177.5785,13.0378,-8135.1948
C00568=-47.238,-63.546,42.745,162.5779,31.0935,-8136.6259
C00569=-49.870,-60.750,42.402,149.8188,28.7683,-8139.3828
C00570=-52.774,-58.195,42.387,149.0312,28.3421,-8142.2032
C00571=-55.552,-55.552,42.397,150.3022,29.6980,-8145.0000
C00572=-58.195,-52.774,42.387,151.6576,30.9686,-8147.7968
C00573=-60.750,-49.870,42.402,151.2308,30.1799,-8150.6172
C00574=-63.546,-47.238,42.745,148.9065,17.4230,-8153.3741
C00575=-66.037,-46.575,43.611,166.9622,-2.4215,-8154.8052
C00576=-68.755,-47.275,44.816,178.2521,-0.7054,-8155.4881
C00577=-71.950,-48.737,46.074,-176.9547,1.4469,-8155.8873
C00578=-75.478,-50.465,47.055,-174.4284,2.4349,-8156.2331
C00579=-79.009,-51.741,47.546,-173.9442,0.8138,-8156.7802
C00580=-82.869,-51.201,47.807,-176.7298,-1.3017,-8158.2900
C00581=-86.517,-48.823,48.020,-178.5970,-1.3527,-8160.5632
C00582=-89.240,-44.981,48.237,-179.9502,-0.0949,-8163.2498
C00583=-91.399,-40.555,48.381,-179.9944,-0.0125,-8166.0725
C00584=-93.306,-35.952,48.381,-179.9951,-0.0128,-8168.9277
C00585=-94.909,-31.296,48.237,-179.9681,-0.1023,-8171.7502
C00586=-95.700,-26.654,48.020,179.9644,-1.9482,-8174.4366
C00587=-94.802,-22.392,47.807,178.6060,-3.2321,-8176.7104
C00588=-92.454,-19.281,47.546,175.1381,-3.7174,-8178.2200
C00589=-89.056,-17.687,47.055,174.3435,-2.2283,-8178.7669
C00590=-85.339,-16.414,46.074,176.8245,-1.1320,-8179.1128
C00591=-82.045,-15.189,44.816,-178.2654,0.7374,-8179.5116
C00592=-79.628,-13.762,43.611,-169.0408,7.6230,-8180.1945
C00593=-78.336,-11.532,42.745,-168.4395,32.9569,-8181.6255
C00594=-78.220,-7.694,42.402,178.6819,38.6410,-8184.3823
C00595=-78.467,-3.833,42.387,177.5412,38.8604,-8187.2034
C00596=-78.562,0.000,42.397,-179.9998,38.8891,-8190.0000
C00597=-78.467,3.833,42.387,-177.5416,38.8604,-8192.7966
C00598=-78.220,7.694,42.402,-178.6839,38.6407,-8195.6177
C00599=-78.336,11.532,42.745,168.4403,32.9573,-8198.3745
C00600=-79.628,13.762,43.611,169.0408,7.6230,-8199.8055
C00601=-82.045,15.189,44.816,178.2654,0.7374,-8200.4884
C00602=-85.339,16.414,46.074,-176.8245,-1.1320,-8200.8872
C00603=-89.056,17.687,47.055,-174.3435,-2.2283,-8201.2331
C00604=-92.454,19.281,47.546,-175.1381,-3.7174,-8201.7800
C00605=-94.802,22.392,47.807,-178.6060,-3.2321,-8203.2896
C00606=-95.700,26.654,48.020,-179.9644,-1.9482,-8205.5634
C00607=-94.909,31.296,48.237,179.9681,-0.1023,-8208.2498
C00608=-93.306,35.952,48.381,179.9951,-0.0128,-8211.0723
C00609=-91.399,40.555,48.381,179.9944,-0.0125,-8213.9275
C00610=-89.240,44.981,48.237,179.9502,-0.0949,-8216.7502
C00611=-86.517,48.823,48.020,178.5970,-1.3527,-8219.4368
C00612=-82.869,51.201,47.807,176.7298,-1.3017,-8221.7100
C00613=-79.009,51.741,47.546,173.9442,0.8138,-8223.2198
C00614=-75.478,50.465,47.055,174.4284,2.4349,-8223.7669
C00615=-71.950,48.737,46.074,176.9547,1.4469,-8224.1127
C00616=-68.755,47.275,44.816,-178.2521,-0.7054,-8224.5119
C00617=-66.037,46.575,43.611,-166.9622,-2.4215,-8225.1948
C00618=-63.546,47.238,42.745,-148.9065,17.4221,-8226.6259
C00619=-60.750,49.870,42.402,-151.2317,30.1812,-8229.3828
C00620=-58.195,52.774,42.387,-151.6579,30.9688,-8232.2032
C00621=-55.552,55.552,42.397,-150.3020,29.6978,-8235.0000
C00622=-52.774,58.195,42.387,-149.0314,28.3424,-8237.7968
C00623=-49.870,60.750,42.402,-149.8201,28.7692,-8240.6172
C00624=-47.238,63.546,42.745,-162.5770,31.0935,-8243.3741
C00625=-46.575,66.037,43.611,177.5785,13.0378,-8244.8052
C00626=-47.275,68.755,44.816,179.2946,1.7479,-8245.4881
C00627=-48.737,71.950,46.074,-178.5531,-3.0453,-8245.8873
C00628=-50.465,75.478,47.055,-177.5651,-5.5716,-8246.2331
C00629=-51.741,79.009,47.546,-179.1862,-6.0558,-8246.7802
C00630=-51.201,82.869,47.807,178.6983,-3.2702,-8248.2900
C00631=-48.823,86.517,48.020,178.6473,-1.4030,-8250.5632
C00632=-44.981,89.240,48.237,179.9051,-0.0498,-8253.2498
C00633=-40.555,91.399,48.381,179.9875,-0.0056,-8256.0725
C00634=-35.952,93.306,48.381,179.9872,-0.0049,-8258.9277
C00635=-31.296,94.909,48.237,179.8977,-0.0319,-8261.7502
C00636=-26.654,95.700,48.020,178.0518,0.0356,-8264.4366
C00637=-22.392,94.802,47.807,176.7679,1.3940,-8266.7104
C00638=-19.281,92.454,47.546,176.2826,4.8619,-8268.2200
C00639=-17.687,89.056,47.055,177.7717,5.6565,-8268.7669
C00640=-16.414,85.339,46.074,178.8680,3.1755,-8269.1128
C00641=-15.189,82.045,44.816,-179.2626,-1.7346,-8269.5116
C00642=-13.762,79.628,43.611,-172.3770,-10.9592,-8270.1945
C00643=-11.532,78.336,42.745,-147.0427,-11.5597,-8271.6255
C00644=-7.694,78.220,42.402,-141.3593,1.3161,-8274.3823
C00645=-3.833,78.467,42.387,-141.1396,2.4584,-8277.2034
C00646=0.000,78.562,42.397,-141.1109,0.0002,-8280.0000
C00647=0.000,77.178,44.107,-140.9045,0.0002,-8280.0000
C00648=3.707,77.088,44.096,-140.9327,-2.4549,-8282.7531
C00649=7.481,76.852,44.112,-141.1728,-1.0178,-8285.5598
C00650=11.270,77.011,44.481,-147.6308,12.5713,-8288.3257
C00651=13.439,78.412,45.416,-173.7657,9.9143,-8289.7254
C00652=14.814,81.004,46.718,-179.6749,0.8332,-8290.3637
C00653=16.001,84.532,48.079,178.7474,-3.8082,-8290.7187
C00654=17.239,88.522,49.141,177.7605,-6.2141,-8291.0200
C00655=18.791,92.187,49.674,176.1706,-5.4532,-8291.5211
C00656=21.929,94.746,49.957,176.4973,-1.6362,-8293.0317
C00657=26.285,95.767,50.188,177.9187,-0.0678,-8295.3479
C00658=31.062,94.986,50.423,179.8864,0.0352,-8298.1086
C00659=35.872,93.336,50.579,179.9859,0.0053,-8301.0234
C00660=40.633,91.364,50.579,179.9863,0.0062,-8303.9765
C00661=45.201,89.129,50.423,179.8948,0.0555,-8306.8914
C00662=49.131,86.304,50.188,178.5759,1.5199,-8309.6519
C00663=51.489,82.502,49.957,178.6776,3.6323,-8311.9680
C00664=51.899,78.473,49.674,-178.8443,6.5508,-8313.4791
C00665=50.405,74.784,49.141,-177.1753,5.9740,-8313.9803
C00666=48.459,71.088,48.079,-178.1897,3.5780,-8314.2813
C00667=46.803,67.754,46.718,179.6407,-0.8190,-8314.6359
C00668=45.943,64.949,45.416,177.3464,-11.3560,-8315.2745
C00669=46.486,62.424,44.481,-163.8001,-31.2115,-8316.6744
C00670=49.053,59.633,44.112,-149.8158,-29.0968,-8319.4401
C00671=51.888,57.130,44.096,-148.8556,-28.5314,-8322.2471
C00672=54.573,54.573,44.107,-150.1203,-29.8799,-8325.0000
C00673=57.130,51.888,44.096,-151.4684,-31.1443,-8327.7529
C00674=59.633,49.053,44.112,-150.9023,-30.1828,-8330.5599
C00675=62.424,46.486,44.482,-148.7885,-16.2008,-8333.3256
C00676=64.949,45.943,45.416,-168.6440,2.6536,-8334.7255
C00677=67.754,46.803,46.718,-179.1810,0.3593,-8335.3641
C00678=71.088,48.459,48.079,176.4220,-1.8103,-8335.7187
C00679=74.784,50.405,49.141,174.0260,-2.8247,-8336.0197
C00680=78.473,51.899,49.674,173.4492,-1.1557,-8336.5209
C00681=82.502,51.489,49.957,176.3677,1.3224,-8338.0320
C00682=86.304,49.131,50.188,178.4801,1.4241,-8340.3481
C00683=89.129,45.201,50.423,179.9445,0.1052,-8343.1086
C00684=91.364,40.633,50.579,179.9938,0.0137,-8346.0235
C00685=93.336,35.872,50.579,179.9947,0.0141,-8348.9766
C00686=94.986,31.062,50.423,179.9648,0.1136,-8351.8914
C00687=95.767,26.285,50.188,-179.9322,2.0813,-8354.6521
C00688=94.746,21.929,49.957,-178.3638,3.5027,-8356.9683
C00689=92.187,18.791,49.674,-174.5468,3.8294,-8358.4789
C00690=88.522,17.239,49.141,-173.7859,2.2395,-8358.9800
C00691=84.532,16.001,48.079,-176.1918,1.2526,-8359.2813
C00692=81.004,14.814,46.718,179.1668,-0.3251,-8359.6363
C00693=78.412,13.439,45.416,170.0857,-6.2343,-8360.2746
C00694=77.011,11.270,44.481,167.4287,-32.3692,-8361.6743
C00695=76.852,7.481,44.112,-178.9822,-38.8272,-8364.4402
C00696=77.088,3.707,44.096,-177.5451,-39.0673,-8367.2469
C00697=77.178,0.000,44.107,179.9998,-39.0955,-8370.0000
C00698=77.088,-3.707,44.096,177.5454,-39.0673,-8372.7531
C00699=76.852,-7.481,44.112,178.9843,-38.8270,-8375.5598
C00700=77.011,-11.270,44.482,-167.4294,-32.3697,-8378.3257
C00701=78.412,-13.439,45.416,-170.0857,-6.2343,-8379.7254
C00702=81.004,-14.814,46.718,-179.1668,-0.3251,-8380.3637
C00703=84.532,-16.001,48.079,176.1918,1.2526,-8380.7187
C00704=88.522,-17.239,49.141,173.7859,2.2395,-8381.0200
C00705=92.187,-18.791,49.674,174.5468,3.8294,-8381.5211
C00706=94.746,-21.929,49.957,178.3638,3.5027,-8383.0317
C00707=95.767,-26.285,50.188,179.9322,2.0813,-8385.3479
C00708=94.986,-31.062,50.423,-179.9648,0.1136,-8388.1086
C00709=93.336,-35.872,50.579,-179.9947,0.0141,-8391.0234
C00710=91.364,-40.633,50.579,-179.9938,0.0137,-8393.9765
C00711=89.129,-45.201,50.423,-179.9445,0.1052,-8396.8914
C00712=86.304,-49.131,50.188,-178.4801,1.4241,-8399.6519
C00713=82.502,-51.489,49.957,-176.3677,1.3224,-8401.9680
C00714=78.473,-51.899,49.674,-173.4492,-1.1557,-8403.4791
C00715=74.784,-50.405,49.141,-174.0260,-2.8247,-8403.9803
C00716=71.088,-48.459,48.079,-176.4220,-1.8103,-8404.2813
C00717=67.754,-46.803,46.718,179.1810,0.3593,-8404.6359
C00718=64.949,-45.943,45.416,168.6440,2.6536,-8405.2745
C00719=62.424,-46.486,44.481,148.7885,-16.1999,-8406.6744
C00720=59.633,-49.053,44.112,150.9032,-30.1842,-8409.4401
C00721=57.130,-51.888,44.096,151.4686,-31.1444,-8412.2471
C00722=54.573,-54.573,44.107,150.1201,-29.8797,-8415.0000
C00723=51.888,-57.130,44.096,148.8557,-28.5316,-8417.7529
C00724=49.053,-59.633,44.112,149.8172,-29.0977,-8420.5599
C00725=46.486,-62.424,44.482,163.7992,-31.2115,-8423.3256
C00726=45.943,-64.949,45.416,-177.3464,-11.3560,-8424.7255
C00727=46.803,-67.754,46.718,-179.6407,-0.8190,-8425.3641
C00728=48.459,-71.088,48.079,178.1897,3.5780,-8425.7187
C00729=50.405,-74.784,49.141,177.1753,5.9740,-8426.0197
C00730=51.899,-78.473,49.674,178.8443,6.5508,-8426.5209
C00731=51.489,-82.502,49.957,-178.6776,3.6323,-8428.0320
C00732=49.131,-86.304,50.188,-178.5759,1.5199,-8430.3481
C00733=45.201,-89.129,50.423,-179.8948,0.0555,-8433.1086
C00734=40.633,-91.364,50.579,-179.9863,0.0062,-8436.0235
C00735=35.872,-93.336,50.579,-179.9859,0.0053,-8438.9766
C00736=31.062,-94.986,50.423,-179.8864,0.0352,-8441.8914
C00737=26.285,-95.767,50.188,-177.9187,-0.0678,-8444.6521
C00738=21.929,-94.746,49.957,-176.4973,-1.6362,-8446.9683
C00739=18.791,-92.187,49.674,-176.1706,-5.4532,-8448.4789
C00740=17.239,-88.522,49.141,-177.7605,-6.2141,-8448.9800
C00741=16.001,-84.532,48.079,-178.7474,-3.8082,-8449.2813
C00742=14.814,-81.004,46.718,179.6749,0.8332,-8449.6363
C00743=13.439,-78.412,45.416,173.7657,9.9143,-8450.2746
C00744=11.270,-77.011,44.481,147.6308,12.5713,-8451.6743
C00745=7.481,-76.852,44.112,141.1728,-1.0178,-8454.4402
C00746=3.707,-77.088,44.096,140.9327,-2.4549,-8457.2469
C00747=0.000,-77.178,44.107,140.9045,0.0002,-8460.0000
C00748=0.000,-77.178,44.107,140.9045,0.0002,-8460.0000
C00749=-3.707,-77.088,44.096,140.9327,2.4546,-8462.7531
C00750=-7.481,-76.852,44.112,141.1730,1.0157,-8465.5598
C00751=-11.270,-77.011,44.482,147.6303,-12.5706,-8468.3257
C00752=-13.439,-78.412,45.416,173.7657,-9.9143,-8469.7254
C00753=-14.814,-81.004,46.718,179.6749,-0.8332,-8470.3637
C00754=-16.001,-84.532,48.079,-178.7474,3.8082,-8470.7187
C00755=-17.239,-88.522,49.141,-177.7605,6.2141,-8471.0200
C00756=-18.791,-92.187,49.674,-176.1706,5.4532,-8471.5211
C00757=-21.929,-94.746,49.957,-176.4973,1.6362,-8473.0317
C00758=-26.285,-95.767,50.188,-177.9187,0.0678,-8475.3479
C00759=-31.062,-94.986,50.423,-179.8864,-0.0352,-8478.1086
C00760=-35.872,-93.336,50.579,-179.9859,-0.0053,-8481.0234
C00761=-40.633,-91.364,50.579,-179.9863,-0.0062,-8483.9765
C00762=-45.201,-89.129,50.423,-179.8948,-0.0555,-8486.8914
C00763=-49.131,-86.304,50.188,-178.5759,-1.5199,-8489.6519
C00764=-51.489,-82.502,49.957,-178.6776,-3.6323,-8491.9680
C00765=-51.899,-78.473,49.674,178.8443,-6.5508,-8493.4791
C00766=-50.405,-74.784,49.141,177.1753,-5.9740,-8493.9803
C00767=-48.459,-71.088,48.079,178.1897,-3.5780,-8494.2813
C00768=-46.803,-67.754,46.718,-179.6407,0.8190,-8494.6359
C00769=-45.943,-64.949,45.416,-177.3464,11.3560,-8495.2745
C00770=-46.486,-62.424,44.481,163.8001,31.2115,-8496.6744
C00771=-49.053,-59.633,44.112,149.8158,29.0968,-8499.4401
C00772=-51.888,-57.130,44.096,148.8556,28.5314,-8502.2471
C00773=-54.573,-54.573,44.107,150.1203,29.8799,-8505.0000
C00774=-57.130,-51.888,44.096,151.4684,31.1443,-8507.7529
C00775=-59.633,-49.053,44.112,150.9023,30.1828,-8510.5599
C00776=-62.424,-46.486,44.482,148.7885,16.2008,-8513.3256
C00777=-64.949,-45.943,45.416,168.6440,-2.6536,-8514.7255
C00778=-67.754,-46.803,46.718,179.1810,-0.3593,-8515.3641
C00779=-71.088,-48.459,48.079,-176.4220,1.8103,-8515.7187
C00780=-74.784,-50.405,49.141,-174.0260,2.8247,-8516.0197
C00781=-78.473,-51.899,49.674,-173.4492,1.1557,-8516.5209
C00782=-82.502,-51.489,49.957,-176.3677,-1.3224,-8518.0320
C00783=-86.304,-49.131,50.188,-178.4801,-1.4241,-8520.3481
C00784=-89.129,-45.201,50.423,-179.9445,-0.1052,-8523.1086
C00785=-91.364,-40.633,50.579,-179.9938,-0.0137,-8526.0235
C00786=-93.336,-35.872,50.579,-179.9947,-0.0141,-8528.9766
C00787=-94.986,-31.062,50.423,-179.9648,-0.1136,-8531.8914
C00788=-95.767,-26.285,50.188,179.9322,-2.0813,-8534.6521
C00789=-94.746,-21.929,49.957,178.3638,-3.5027,-8536.9683
C00790=-92.187,-18.791,49.674,174.5468,-3.8294,-8538.4789
C00791=-88.522,-17.239,49.141,173.7859,-2.2395,-8538.9800
C00792=-84.532,-16.001,48.079,176.1918,-1.2526,-8539.2813
C00793=-81.004,-14.814,46.718,-179.1668,0.3251,-8539.6363
C00794=-78.412,-13.439,45.416,-170.0857,6.2343,-8540.2746
C00795=-77.011,-11.270,44.481,-167.4287,32.3692,-8541.6743
C00796=-76.852,-7.481,44.112,178.9822,38.8272,-8544.4402
C00797=-77.088,-3.707,44.096,177.5451,39.0673,-8547.2469
C00798=-77.178,0.000,44.107,-179.9998,39.0955,-8550.0000
C00799=-77.088,3.707,44.096,-177.5454,39.0673,-8552.7531
C00800=-76.852,7.481,44.112,-178.9843,38.8270,-8555.5598
C00801=-77.011,11.270,44.482,167.4294,32.3697,-8558.3257
C00802=-78.412,13.439,45.416,170.0857,6.2343,-8559.7254
C00803=-81.004,14.814,46.718,179.1668,0.3251,-8560.3637
C00804=-84.532,16.001,48.079,-176.1918,-1.2526,-8560.7187
C00805=-88.522,17.239,49.141,-173.7859,-2.2395,-8561.0200
C00806=-92.187,18.791,49.674,-174.5468,-3.8294,-8561.5211
C00807=-94.746,21.929,49.957,-178.3638,-3.5027,-8563.0317
C00808=-95.767,26.285,50.188,-179.9322,-2.0813,-8565.3479
C00809=-94.986,31.062,50.423,179.9648,-0.1136,-8568.1086
C00810=-93.336,35.872,50.579,179.9947,-0.0141,-8571.0234
C00811=-91.364,40.633,50.579,179.9938,-0.0137,-8573.9765
C00812=-89.129,45.201,50.423,179.9445,-0.1052,-8576.8914
C00813=-86.304,49.131,50.188,178.4801,-1.4241,-8579.6519
C00814=-82.502,51.489,49.957,176.3677,-1.3224,-8581.9680
C00815=-78.473,51.899,49.674,173.4492,1.1557,-8583.4791
C00816=-74.784,50.405,49.141,174.0260,2.8247,-8583.9803
C00817=-71.088,48.459,48.079,176.4220,1.8103,-8584.2813
C00818=-67.754,46.803,46.718,-179.1810,-0.3593,-8584.6359
C00819=-64.949,45.943,45.416,-168.6440,-2.6536,-8585.2745
C00820=-62.424,46.486,44.481,-148.7885,16.1999,-8586.6744
C00821=-59.633,49.053,44.112,-150.9032,30.1842,-8589.4401
C00822=-57.130,51.888,44.096,-151.4686,31.1444,-8592.2471
C00823=-54.573,54.573,44.107,-150.1201,29.8797,-8595.0000
C00824=-51.888,57.130,44.096,-148.8557,28.5316,-8597.7529
C00825=-49.053,59.633,44.112,-149.8172,29.0977,-8600.5599
C00826=-46.486,62.424,44.482,-163.7992,31.2115,-8603.3256
C00827=-45.943,64.949,45.416,177.3464,11.3560,-8604.7255
C00828=-46.803,67.754,46.718,179.6407,0.8190,-8605.3641
C00829=-48.459,71.088,48.079,-178.1897,-3.5780,-8605.7187
C00830=-50.405,74.784,49.141,-177.1753,-5.9740,-8606.0197
C00831=-51.899,78.473,49.674,-178.8443,-6.5508,-8606.5209
C00832=-51.489,82.502,49.957,178.6776,-3.6323,-8608.0320
C00833=-49.131,86.304,50.188,178.5759,-1.5199,-8610.3481
C00834=-45.201,89.129,50.423,179.8948,-0.0555,-8613.1086
C00835=-40.633,91.364,50.579,179.9863,-0.0062,-8616.0235
C00836=-35.872,93.336,50.579,179.9859,-0.0053,-8618.9766
C00837=-31.062,94.986,50.423,179.8864,-0.0352,-8621.8914
C00838=-26.285,95.767,50.188,177.9187,0.0678,-8624.6521
C00839=-21.929,94.746,49.957,176.4973,1.6362,-8626.9683
C00840=-18.791,92.187,49.674,176.1706,5.4532,-8628.4789
C00841=-17.239,88.522,49.141,177.7605,6.2141,-8628.9800
C00842=-16.001,84.532,48.079,178.7474,3.8082,-8629.2813
C00843=-14.814,81.004,46.718,-179.6749,-0.8332,-8629.6363
C00844=-13.439,78.412,45.416,-173.7657,-9.9143,-8630.2746
C00845=-11.270,77.011,44.482,-147.6303,-12.5706,-8631.6743
C00846=-7.481,76.852,44.112,-141.1730,1.0157,-8634.4402
C00847=-3.707,77.088,44.096,-140.9327,2.4546,-8637.2469
C00848=0.000,77.178,44.107,-140.9045,0.0002,-8640.0000
C00849=0.000,75.789,45.812,-140.7733,0.0001,-8640.0000
C00850=3.580,75.703,45.801,-140.8009,-2.4427,-8642.7075
C00851=7.267,75.480,45.818,-141.0649,-0.7003,-8645.4993
C00852=11.008,75.681,46.215,-148.3523,13.4833,-8648.2758
C00853=13.116,77.193,47.218,-174.9743,8.8067,-8649.6431
C00854=14.439,79.961,48.618,-179.9989,0.0032,-8650.2359
C00855=15.588,83.726,50.084,178.6708,-4.3591,-8650.5465
C00856=16.791,87.989,51.229,177.7869,-6.6807,-8650.8039
C00857=18.302,91.921,51.802,176.1277,-5.9675,-8651.2607
C00858=21.467,94.690,52.107,176.2739,-1.8689,-8652.7735
C00859=25.919,95.834,52.356,177.8036,-0.1013,-8655.1340
C00860=30.830,95.062,52.610,179.8764,0.0380,-8657.9686
C00861=35.794,93.367,52.777,179.9849,0.0057,-8660.9753
C00862=40.710,91.330,52.777,179.9853,0.0067,-8664.0247
C00863=45.419,89.019,52.610,179.8857,0.0605,-8667.0314
C00864=49.437,86.092,52.356,178.5181,1.6250,-8669.8659
C00865=51.776,82.136,52.107,178.6837,3.9541,-8672.2261
C00866=52.057,77.939,51.802,-178.5076,6.9431,-8673.7397
C00867=50.345,74.091,51.229,-176.8234,6.2858,-8674.1962
C00868=48.181,70.226,50.084,-177.8528,4.0217,-8674.4534
C00869=46.331,66.751,48.618,179.9986,-0.0031,-8674.7640
C00870=45.309,63.858,47.218,177.2881,-9.7446,-8675.3567
C00871=45.731,61.299,46.215,-165.0891,-31.1895,-8676.7241
C00872=48.234,58.511,45.818,-149.8897,-29.3636,-8679.5007
C00873=50.999,56.061,45.801,-148.7486,-28.6575,-8682.2930
C00874=53.591,53.591,45.812,-150.0043,-29.9958,-8685.0000
C00875=56.061,50.999,45.801,-151.3424,-31.2514,-8687.7070
C00876=58.511,48.233,45.818,-150.6354,-30.1089,-8690.4999
C00877=61.299,45.731,46.215,-148.8104,-14.9118,-8693.2759
C00878=63.858,45.309,47.218,-170.2554,2.7119,-8694.6433
C00879=66.751,46.331,48.618,-179.9969,0.0014,-8695.2360
C00880=70.226,48.181,50.084,175.9783,-2.1472,-8695.5466
C00881=74.091,50.345,51.229,173.7142,-3.1766,-8695.8038
C00882=77.939,52.057,51.802,173.0569,-1.4924,-8696.2603
C00883=82.136,51.776,52.107,176.0459,1.3163,-8697.7739
C00884=86.092,49.437,52.356,178.3750,1.4819,-8700.1341
C00885=89.019,45.419,52.610,179.9395,0.1143,-8702.9686
C00886=91.330,40.710,52.777,179.9933,0.0147,-8705.9753
C00887=93.367,35.794,52.777,179.9943,0.0151,-8709.0247
C00888=95.062,30.830,52.610,179.9620,0.1236,-8712.0314
C00889=95.834,25.919,52.356,-179.8987,2.1964,-8714.8660
C00890=94.690,21.467,52.107,-178.1311,3.7261,-8717.2265
C00891=91.921,18.302,51.802,-174.0325,3.8723,-8718.7393
C00892=87.989,16.791,51.229,-173.3193,2.2131,-8719.1961
C00893=83.726,15.588,50.084,-175.6409,1.3292,-8719.4535
C00894=79.961,14.439,48.618,179.9968,-0.0011,-8719.7641
C00895=77.193,13.116,47.218,171.1933,-5.0257,-8720.3569
C00896=75.681,11.008,46.215,166.5167,-31.6477,-8721.7242
C00897=75.480,7.267,45.818,-179.2997,-38.9351,-8724.5007
C00898=75.703,3.580,45.801,-177.5573,-39.1991,-8727.2925
C00899=75.789,0.000,45.812,179.9999,-39.2267,-8730.0000
C00900=75.703,-3.580,45.801,177.5575,-39.1992,-8732.7075
C00901=75.480,-7.267,45.818,179.3020,-38.9348,-8735.4993
C00902=75.681,-11.008,46.215,-166.5172,-31.6482,-8738.2758
C00903=77.193,-13.116,47.218,-171.1933,-5.0257,-8739.6431
C00904=79.961,-14.439,48.618,-179.9968,-0.0011,-8740.2359
C00905=83.726,-15.588,50.084,175.6409,1.3292,-8740.5465
C00906=87.989,-16.791,51.229,173.3193,2.2131,-8740.8039
C00907=91.921,-18.302,51.802,174.0325,3.8723,-8741.2607
C00908=94.690,-21.467,52.107,178.1311,3.7261,-8742.7735
C00909=95.834,-25.919,52.356,179.8987,2.1964,-8745.1340
C00910=95.062,-30.830,52.610,-179.9620,0.1236,-8747.9686
C00911=93.367,-35.794,52.777,-179.9943,0.0151,-8750.9753
C00912=91.330,-40.710,52.777,-179.9933,0.0147,-8754.0247
C00913=89.019,-45.419,52.610,-179.9395,0.1143,-8757.0314
C00914=86.092,-49.437,52.356,-178.3750,1.4819,-8759.8659
C00915=82.136,-51.776,52.107,-176.0459,1.3163,-8762.2261
C00916=77.939,-52.057,51.802,-173.0569,-1.4924,-8763.7397
C00917=74.091,-50.345,51.229,-173.7142,-3.1766,-8764.1962
C00918=70.226,-48.181,50.084,-175.9783,-2.1472,-8764.4534
C00919=66.751,-46.331,48.618,179.9969,0.0014,-8764.7640
C00920=63.858,-45.309,47.218,170.2554,2.7119,-8765.3567
C00921=61.299,-45.731,46.215,148.8105,-14.9109,-8766.7241
C00922=58.511,-48.234,45.818,150.6364,-30.1103,-8769.5007
C00923=56.061,-50.999,45.801,151.3425,-31.2514,-8772.2930
C00924=53.591,-53.591,45.812,150.0042,-29.9957,-8775.0000
C00925=50.999,-56.061,45.801,148.7486,-28.6576,-8777.7070
C00926=48.233,-58.511,45.818,149.8911,-29.3646,-8780.4999
C00927=45.731,-61.299,46.215,165.0882,-31.1896,-8783.2759
C00928=45.309,-63.858,47.218,-177.2881,-9.7446,-8784.6433
C00929=46.331,-66.751,48.618,-179.9986,-0.0031,-8785.2360
C00930=48.181,-70.226,50.084,177.8528,4.0217,-8785.5466
C00931=50.345,-74.091,51.229,176.8234,6.2858,-8785.8038
C00932=52.057,-77.939,51.802,178.5076,6.9431,-8786.2603
C00933=51.776,-82.136,52.107,-178.6837,3.9541,-8787.7739
C00934=49.437,-86.092,52.356,-178.5181,1.6250,-8790.1341
C00935=45.419,-89.019,52.610,-179.8857,0.0605,-8792.9686
C00936=40.710,-91.330,52.777,-179.9853,0.0067,-8795.9753
C00937=35.794,-93.367,52.777,-179.9849,0.0057,-8799.0247
C00938=30.830,-95.062,52.610,-179.8764,0.0380,-8802.0314
C00939=25.919,-95.834,52.356,-177.8036,-0.1013,-8804.8660
C00940=21.467,-94.690,52.107,-176.2739,-1.8689,-8807.2265
C00941=18.302,-91.921,51.802,-176.1277,-5.9675,-8808.7393
C00942=16.791,-87.989,51.229,-177.7869,-6.6807,-8809.1961
C00943=15.588,-83.726,50.084,-178.6708,-4.3591,-8809.4535
C00944=14.439,-79.961,48.618,179.9989,0.0032,-8809.7641
C00945=13.116,-77.193,47.218,174.9743,8.8067,-8810.3569
C00946=11.008,-75.681,46.215,148.3523,13.4833,-8811.7242
C00947=7.267,-75.480,45.818,141.0649,-0.7003,-8814.5007
C00948=3.580,-75.703,45.801,140.8009,-2.4427,-8817.2925
C00949=0.000,-75.789,45.812,140.7733,0.0001,-8820.0000
C00950=0.000,-75.789,45.812,140.7733,0.0001,-8820.0000
C00951=-3.580,-75.703,45.801,140.8008,2.4425,-8822.7075
C00952=-7.267,-75.480,45.818,141.0652,0.6980,-8825.4993
C00953=-11.008,-75.681,46.215,148.3518,-13.4828,-8828.2758
C00954=-13.116,-77.193,47.218,174.9743,-8.8067,-8829.6431
C00955=-14.439,-79.961,48.618,179.9989,-0.0032,-8830.2359
C00956=-15.588,-83.726,50.084,-178.6708,4.3591,-8830.5465
C00957=-16.791,-87.989,51.229,-177.7869,6.6807,-8830.8039
C00958=-18.302,-91.921,51.802,-176.1277,5.9675,-8831.2607
C00959=-21.467,-94.690,52.107,-176.2739,1.8689,-8832.7735
C00960=-25.919,-95.834,52.356,-177.8036,0.1013,-8835.1340
C00961=-30.830,-95.062,52.610,-179.8764,-0.0380,-8837.9686
C00962=-35.794,-93.367,52.777,-179.9849,-0.0057,-8840.9753
C00963=-40.710,-91.330,52.777,-179.9853,-0.0067,-8844.0247
C00964=-45.419,-89.019,52.610,-179.8857,-0.0605,-8847.0314
C00965=-49.437,-86.092,52.356,-178.5181,-1.6250,-8849.8659
C00966=-51.776,-82.136,52.107,-178.6837,-3.9541,-8852.2261
C00967=-52.057,-77.939,51.802,178.5076,-6.9431,-8853.7397
C00968=-50.345,-74.091,51.229,176.8234,-6.2858,-8854.1962
C00969=-48.181,-70.226,50.084,177.8528,-4.0217,-8854.4534
C00970=-46.331,-66.751,48.618,-179.9986,0.0031,-8854.7640
C00971=-45.309,-63.858,47.218,-177.2881,9.7446,-8855.3567
C00972=-45.731,-61.299,46.215,165.0891,31.1895,-8856.7241
C00973=-48.234,-58.511,45.818,149.8897,29.3636,-8859.5007
C00974=-50.999,-56.061,45.801,148.7486,28.6575,-8862.2930
C00975=-53.591,-53.591,45.812,150.0043,29.9958,-8865.0000
C00976=-56.061,-50.999,45.801,151.3424,31.2514,-8867.7070
C00977=-58.511,-48.233,45.818,150.6354,30.1089,-8870.4999
C00978=-61.299,-45.731,46.215,148.8104,14.9118,-8873.2759
C00979=-63.858,-45.309,47.218,170.2554,-2.7119,-8874.6433
C00980=-66.751,-46.331,48.618,179.9969,-0.0014,-8875.2360
C00981=-70.226,-48.181,50.084,-175.9783,2.1472,-8875.5466
C00982=-74.091,-50.345,51.229,-173.7142,3.1766,-8875.8038
C00983=-77.939,-52.057,51.802,-173.0569,1.4924,-8876.2603
C00984=-82.136,-51.776,52.107,-176.0459,-1.3163,-8877.7739
C00985=-86.092,-49.437,52.356,-178.3750,-1.4819,-8880.1341
C00986=-89.019,-45.419,52.610,-179.9395,-0.1143,-8882.9686
C00987=-91.330,-40.710,52.777,-179.9933,-0.0147,-8885.9753
C00988=-93.367,-35.794,52.777,-179.9943,-0.0151,-8889.0247
C00989=-95.062,-30.830,52.610,-179.9620,-0.1236,-8892.0314
C00990=-95.834,-25.919,52.356,179.8987,-2.1964,-8894.8660
C00991=-94.690,-21.467,52.107,178.1311,-3.7261,-8897.2265
C00992=-91.921,-18.302,51.802,174.0325,-3.8723,-8898.7393
C00993=-87.989,-16.791,51.229,173.3193,-2.2131,-8899.1961
C00994=-83.726,-15.588,50.084,175.6409,-1.3292,-8899.4535
C00995=-79.961,-14.439,48.618,-179.9968,0.0011,-8899.7641
C00996=-77.193,-13.116,47.218,-171.1933,5.0257,-8900.3569
C00997=-75.681,-11.008,46.215,-166.5167,31.6477,-8901.7242
C00998=-75.480,-7.267,45.818,179.2997,38.9351,-8904.5007
C00999=-75.703,-3.580,45.801,177.5573,39.1991,-8907.2925
C01000=-75.789,0.000,45.812,-179.9999,39.2267,-8910.0000
C01001=-75.703,3.580,45.801,-177.5575,39.1992,-8912.7075
C01002=-75.480,7.267,45.818,-179.3020,38.9348,-8915.4993
C01003=-75.681,11.008,46.215,166.5172,31.6482,-8918.2758
C01004=-77.193,13.116,47.218,171.1933,5.0257,-8919.6431
C01005=-79.961,14.439,48.618,179.9968,0.0011,-8920.2359
C01006=-83.726,15.588,50.084,-175.6409,-1.3292,-8920.5465
C01007=-87.989,16.791,51.229,-173.3193,-2.2131,-8920.8039
C01008=-91.921,18.302,51.802,-174.0325,-3.8723,-8921.2607
C01009=-94.690,21.467,52.107,-178.1311,-3.7261,-8922.7735
C01010=-95.834,25.919,52.356,-179.8987,-2.1964,-8925.1340
C01011=-95.062,30.830,52.610,179.9620,-0.1236,-8927.9686
C01012=-93.367,35.794,52.777,179.9943,-0.0151,-8930.9753
C01013=-91.330,40.710,52.777,179.9933,-0.0147,-8934.0247
C01014=-89.019,45.419,52.610,179.9395,-0.1143,-8937.0314
C01015=-86.092,49.437,52.356,178.3750,-1.4819,-8939.8659
C01016=-82.136,51.776,52.107,176.0459,-1.3163,-8942.2261
C01017=-77.939,52.057,51.802,173.0569,1.4924,-8943.7397
C01018=-74.091,50.345,51.229,173.7142,3.1766,-8944.1962
C01019=-70.226,48.181,50.084,175.9783,2.1472,-8944.4534
C01020=-66.751,46.331,48.618,-179.9969,-0.0014,-8944.7640
C01021=-63.858,45.309,47.218,-170.2554,-2.7119,-8945.3567
C01022=-61.299,45.731,46.215,-148.8105,14.9109,-8946.7241
C01023=-58.511,48.234,45.818,-150.6364,30.1103,-8949.5007
C01024=-56.061,50.999,45.801,-151.3425,31.2514,-8952.2930
C01025=-53.591,53.591,45.812,-150.0042,29.9957,-8955.0000
C01026=-50.999,56.061,45.801,-148.7486,28.6576,-8957.7070
C01027=-48.233,58.511,45.818,-149.8911,29.3646,-8960.4999
C01028=-45.731,61.299,46.215,-165.0882,31.1896,-8963.2759
C01029=-45.309,63.858,47.218,177.2881,9.7446,-8964.6433
C01030=-46.331,66.751,48.618,179.9986,0.0031,-8965.2360
C01031=-48.181,70.226,50.084,-177.8528,-4.0217,-8965.5466
C01032=-50.345,74.091,51.229,-176.8234,-6.2858,-8965.8038
C01033=-52.057,77.939,51.802,-178.5076,-6.9431,-8966.2603
C01034=-51.776,82.136,52.107,178.6837,-3.9541,-8967.7739
C01035=-49.437,86.092,52.356,178.5181,-1.6250,-8970.1341
C01036=-45.419,89.019,52.610,179.8857,-0.0605,-8972.9686
C01037=-40.710,91.330,52.777,179.9853,-0.0067,-8975.9753
C01038=-35.794,93.367,52.777,179.9849,-0.0057,-8979.0247
C01039=-30.830,95.062,52.610,179.8764,-0.0380,-8982.0314
C01040=-25.919,95.834,52.356,177.8036,0.1013,-8984.8660
C01041=-21.467,94.690,52.107,176.2739,1.8689,-8987.2265
C01042=-18.302,91.921,51.802,176.1277,5.9675,-8988.7393
C01043=-16.791,87.989,51.229,177.7869,6.6807,-8989.1961
C01044=-15.588,83.726,50.084,178.6708,4.3591,-8989.4535
C01045=-14.439,79.961,48.618,-179.9989,-0.0032,-8989.7641
C01046=-13.116,77.193,47.218,-174.9743,-8.8067,-8990.3569
C01047=-11.008,75.681,46.215,-148.3518,-13.4828,-8991.7242
C01048=-7.267,75.480,45.818,-141.0652,0.6980,-8994.5007
C01049=-3.580,75.703,45.801,-140.8008,2.4425,-8997.2925
C01050=0.000,75.789,45.812,-140.7733,0.0001,-9000.0000
C01051=0.000,74.396,47.516,-140.7158,0.0000,-9000.0000
C01052=3.453,74.315,47.503,-140.7427,-2.4223,-9002.6603
C01053=7.053,74.105,47.522,-141.0345,-0.3681,-9005.4368
C01054=10.745,74.349,47.946,-149.1996,14.2839,-9008.2235
C01055=12.792,75.972,49.019,-176.0111,7.6747,-9009.5577
C01056=14.064,78.919,50.519,179.7498,-0.7514,-9010.1045
C01057=15.177,82.922,52.090,178.6288,-4.8303,-9010.3719
C01058=16.346,87.459,53.317,177.8411,-7.0591,-9010.5864
C01059=17.816,91.657,53.931,176.1414,-6.4001,-9010.9998
C01060=21.009,94.635,54.258,176.0979,-2.0860,-9012.5167
C01061=25.555,95.900,54.525,177.7079,-0.1349,-9014.9212
C01062=30.600,95.138,54.796,179.8678,0.0404,-9017.8298
C01063=35.715,93.397,54.976,179.9840,0.0060,-9020.9268
C01064=40.787,91.296,54.976,179.9844,0.0071,-9024.0730
C01065=45.636,88.910,54.796,179.8779,0.0649,-9027.1707
C01066=49.741,85.881,54.525,178.4742,1.7165,-9030.0788
C01067=52.061,81.773,54.258,178.7124,4.2314,-9032.4830
C01068=52.213,77.409,53.931,-178.1887,7.2383,-9034.0000
C01069=50.285,73.401,53.317,-176.5147,6.5160,-9034.4140
C01070=47.903,69.367,52.090,-177.5476,4.3848,-9034.6279
C01071=45.859,65.749,50.519,-179.6456,0.7082,-9034.8952
C01072=44.675,62.766,49.019,177.3675,-8.2277,-9035.4421
C01073=44.975,60.171,47.946,-166.4231,-31.0292,-9036.7764
C01074=47.412,57.387,47.522,-150.0390,-29.5687,-9039.5628
C01075=50.108,54.990,47.503,-148.7091,-28.7213,-9042.3404
C01076=52.606,52.606,47.516,-149.9535,-30.0466,-9045.0000
C01077=54.990,50.108,47.503,-151.2786,-31.2909,-9047.6596
C01078=57.387,47.412,47.522,-150.4303,-29.9595,-9050.4372
C01079=60.171,44.975,47.946,-148.9707,-13.5777,-9053.2236
C01080=62.766,44.675,49.019,-171.7723,2.6325,-9054.5579
C01081=65.749,45.859,50.519,179.2918,-0.3544,-9055.1048
C01082=69.367,47.903,52.090,175.6152,-2.4524,-9055.3721
C01083=73.401,50.285,53.317,173.4840,-3.4853,-9055.5860
C01084=77.409,52.213,53.931,172.7617,-1.8113,-9056.0000
C01085=81.773,52.061,54.258,175.7686,1.2876,-9057.5170
C01086=85.881,49.741,54.525,178.2835,1.5258,-9059.9212
C01087=88.910,45.636,54.796,179.9351,0.1221,-9062.8293
C01088=91.296,40.787,54.976,179.9929,0.0156,-9065.9270
C01089=93.397,35.715,54.976,179.9940,0.0160,-9069.0732
C01090=95.138,30.600,54.796,179.9596,0.1322,-9072.1702
C01091=95.900,25.555,54.525,-179.8651,2.2921,-9075.0788
C01092=94.635,21.009,54.258,-177.9140,3.9021,-9077.4833
C01093=91.657,17.816,53.931,-173.5999,3.8586,-9079.0002
C01094=87.459,16.346,53.317,-172.9409,2.1589,-9079.4136
C01095=82.922,15.177,52.090,-175.1697,1.3712,-9079.6281
C01096=78.919,14.064,50.519,-179.2486,0.2502,-9079.8955
C01097=75.972,12.792,49.019,172.3253,-3.9889,-9080.4423
C01098=74.349,10.745,47.946,165.7161,-30.8004,-9081.7765
C01099=74.105,7.053,47.522,-179.6319,-38.9655,-9084.5632
C01100=74.315,3.453,47.503,-177.5777,-39.2573,-9087.3397
C01101=74.396,0.000,47.516,180.0000,-39.2842,-9090.0000
C01102=74.315,-3.453,47.503,177.5778,-39.2573,-9092.6603
C01103=74.105,-7.053,47.522,179.6343,-38.9652,-9095.4368
C01104=74.349,-10.745,47.946,-165.7166,-30.8009,-9098.2235
C01105=75.972,-12.792,49.019,-172.3253,-3.9889,-9099.5577
C01106=78.919,-14.064,50.519,179.2486,0.2502,-9100.1045
C01107=82.922,-15.177,52.090,175.1697,1.3712,-9100.3719
C01108=87.459,-16.346,53.317,172.9409,2.1589,-9100.5864
C01109=91.657,-17.816,53.931,173.5999,3.8586,-9100.9998
C01110=94.635,-21.009,54.258,177.9140,3.9021,-9102.5167
C01111=95.900,-25.555,54.525,179.8651,2.2921,-9104.9212
C01112=95.138,-30.600,54.796,-179.9596,0.1322,-9107.8298
C01113=93.397,-35.715,54.976,-179.9940,0.0160,-9110.9268
C01114=91.296,-40.787,54.976,-179.9929,0.0156,-9114.0730
C01115=88.910,-45.636,54.796,-179.9351,0.1221,-9117.1707
C01116=85.881,-49.741,54.525,-178.2835,1.5258,-9120.0788
C01117=81.773,-52.061,54.258,-175.7686,1.2876,-9122.4830
C01118=77.409,-52.213,53.931,-172.7617,-1.8113,-9124.0000
C01119=73.401,-50.285,53.317,-173.4840,-3.4853,-9124.4140
C01120=69.367,-47.903,52.090,-175.6152,-2.4524,-9124.6279
C01121=65.749,-45.859,50.519,-179.2918,-0.3544,-9124.8952
C01122=62.766,-44.675,49.019,171.7723,2.6325,-9125.4421
C01123=60.171,-44.975,47.946,148.9708,-13.5769,-9126.7764
C01124=57.387,-47.412,47.522,150.4313,-29.9610,-9129.5628
C01125=54.990,-50.108,47.503,151.2787,-31.2909,-9132.3404
C01126=52.606,-52.606,47.516,149.9534,-30.0465,-9135.0000
C01127=50.108,-54.990,47.503,148.7091,-28.7214,-9137.6596
C01128=47.412,-57.387,47.522,150.0405,-29.5697,-9140.4372
C01129=44.975,-60.171,47.946,166.4223,-31.0293,-9143.2236
C01130=44.675,-62.766,49.019,-177.3675,-8.2277,-9144.5579
C01131=45.859,-65.749,50.519,179.6456,0.7082,-9145.1048
C01132=47.903,-69.367,52.090,177.5476,4.3848,-9145.3721
C01133=50.285,-73.401,53.317,176.5147,6.5160,-9145.5860
C01134=52.213,-77.409,53.931,178.1887,7.2383,-9146.0000
C01135=52.061,-81.773,54.258,-178.7124,4.2314,-9147.5170
C01136=49.741,-85.881,54.525,-178.4742,1.7165,-9149.9212
C01137=45.636,-88.910,54.796,-179.8779,0.0649,-9152.8293
C01138=40.787,-91.296,54.976,-179.9844,0.0071,-9155.9270
C01139=35.715,-93.397,54.976,-179.9840,0.0060,-9159.0732
C01140=30.600,-95.138,54.796,-179.8678,0.0404,-9162.1702
C01141=25.555,-95.900,54.525,-177.7079,-0.1349,-9165.0788
C01142=21.009,-94.635,54.258,-176.0979,-2.0860,-9167.4833
C01143=17.816,-91.657,53.931,-176.1414,-6.4001,-9169.0002
C01144=16.346,-87.459,53.317,-177.8411,-7.0591,-9169.4136
C01145=15.177,-82.922,52.090,-178.6288,-4.8303,-9169.6281
C01146=14.064,-78.919,50.519,-179.7498,-0.7514,-9169.8955
C01147=12.792,-75.972,49.019,176.0111,7.6747,-9170.4423
C01148=10.745,-74.349,47.946,149.1996,14.2839,-9171.7765
C01149=7.053,-74.105,47.522,141.0345,-0.3681,-9174.5632
C01150=3.453,-74.315,47.503,140.7427,-2.4223,-9177.3397
C01151=0.000,-74.396,47.516,140.7158,0.0000,-9180.0000
C01152=0.000,-74.396,47.516,140.7158,0.0000,-9180.0000
C01153=-3.453,-74.315,47.503,140.7427,2.4222,-9182.6603
C01154=-7.053,-74.105,47.522,141.0348,0.3657,-9185.4368
C01155=-10.745,-74.349,47.946,149.1991,-14.2834,-9188.2235
C01156=-12.792,-75.972,49.019,176.0111,-7.6747,-9189.5577
C01157=-14.064,-78.919,50.519,-179.7498,0.7514,-9190.1045
C01158=-15.177,-82.922,52.090,-178.6288,4.8303,-9190.3719
C01159=-16.346,-87.459,53.317,-177.8411,7.0591,-9190.5864
C01160=-17.816,-91.657,53.931,-176.1414,6.4001,-9190.9998
C01161=-21.009,-94.635,54.258,-176.0979,2.0860,-9192.5167
C01162=-25.555,-95.900,54.525,-177.7079,0.1349,-9194.9212
C01163=-30.600,-95.138,54.796,-179.8678,-0.0404,-9197.8298
C01164=-35.715,-93.397,54.976,-179.9840,-0.0060,-9200.9268
C01165=-40.787,-91.296,54.976,-179.9844,-0.0071,-9204.0730
C01166=-45.636,-88.910,54.796,-179.8779,-0.0649,-9207.1707
C01167=-49.741,-85.881,54.525,-178.4742,-1.7165,-9210.0788
C01168=-52.061,-81.773,54.258,-178.7124,-4.2314,-9212.4830
C01169=-52.213,-77.409,53.931,178.1887,-7.2383,-9214.0000
C01170=-50.285,-73.401,53.317,176.5147,-6.5160,-9214.4140
C01171=-47.903,-69.367,52.090,177.5476,-4.3848,-9214.6279
C01172=-45.859,-65.749,50.519,179.6456,-0.7082,-9214.8952
C01173=-44.675,-62.766,49.019,-177.3675,8.2277,-9215.4421
C01174=-44.975,-60.171,47.946,166.4231,31.0292,-9216.7764
C01175=-47.412,-57.387,47.522,150.0390,29.5687,-9219.5628
C01176=-50.108,-54.990,47.503,148.7091,28.7213,-9222.3404
C01177=-52.606,-52.606,47.516,149.9535,30.0466,-9225.0000
C01178=-54.990,-50.108,47.503,151.2786,31.2909,-9227.6596
C01179=-57.387,-47.412,47.522,150.4303,29.9595,-9230.4372
C01180=-60.171,-44.975,47.946,148.9707,13.5777,-9233.2236
C01181=-62.766,-44.675,49.019,171.7723,-2.6325,-9234.5579
C01182=-65.749,-45.859,50.519,-179.2918,0.3544,-9235.1048
C01183=-69.367,-47.903,52.090,-175.6152,2.4524,-9235.3721
C01184=-73.401,-50.285,53.317,-173.4840,3.4853,-9235.5860
C01185=-77.409,-52.213,53.931,-172.7617,1.8113,-9236.0000
C01186=-81.773,-52.061,54.258,-175.7686,-1.2876,-9237.5170
C01187=-85.881,-49.741,54.525,-178.2835,-1.5258,-9239.9212
C01188=-88.910,-45.636,54.796,-179.9351,-0.1221,-9242.8293
C01189=-91.296,-40.787,54.976,-179.9929,-0.0156,-9245.9270
C01190=-93.397,-35.715,54.976,-179.9940,-0.0160,-9249.0732
C01191=-95.138,-30.600,54.796,-179.9596,-0.1322,-9252.1702
C01192=-95.900,-25.555,54.525,179.8651,-2.2921,-9255.0788
C01193=-94.635,-21.009,54.258,177.9140,-3.9021,-9257.4833
C01194=-91.657,-17.816,53.931,173.5999,-3.8586,-9259.0002
C01195=-87.459,-16.346,53.317,172.9409,-2.1589,-9259.4136
C01196=-82.922,-15.177,52.090,175.1697,-1.3712,-9259.6281
C01197=-78.919,-14.064,50.519,179.2486,-0.2502,-9259.8955
C01198=-75.972,-12.792,49.019,-172.3253,3.9889,-9260.4423
C01199=-74.349,-10.745,47.946,-165.7161,30.8004,-9261.7765
C01200=-74.105,-7.053,47.522,179.6319,38.9655,-9264.5632
C01201=-74.315,-3.453,47.503,177.5777,39.2573,-9267.3397
C01202=-74.396,0.000,47.516,-180.0000,39.2842,-9270.0000
C01203=-74.315,3.453,47.503,-177.5778,39.2573,-9272.6603
C01204=-74.105,7.053,47.522,-179.6343,38.9652,-9275.4368
C01205=-74.349,10.745,47.946,165.7166,30.8009,-9278.2235
C01206=-75.972,12.792,49.019,172.3253,3.9889,-9279.5577
C01207=-78.919,14.064,50.519,-179.2486,-0.2502,-9280.1045
C01208=-82.922,15.177,52.090,-175.1697,-1.3712,-9280.3719
C01209=-87.459,16.346,53.317,-172.9409,-2.1589,-9280.5864
C01210=-91.657,17.816,53.931,-173.5999,-3.8586,-9280.9998
C01211=-94.635,21.009,54.258,-177.9140,-3.9021,-9282.5167
C01212=-95.900,25.555,54.525,-179.8651,-2.2921,-9284.9212
C01213=-95.138,30.600,54.796,179.9596,-0.1322,-9287.8298
C01214=-93.397,35.715,54.976,179.9940,-0.0160,-9290.9268
C01215=-91.296,40.787,54.976,179.9929,-0.0156,-9294.0730
C01216=-88.910,45.636,54.796,179.9351,-0.1221,-9297.1707
C01217=-85.881,49.741,54.525,178.2835,-1.5258,-9300.0788
C01218=-81.773,52.061,54.258,175.7686,-1.2876,-9302.4830
C01219=-77.409,52.213,53.931,172.7617,1.8113,-9304.0000
C01220=-73.401,50.285,53.317,173.4840,3.4853,-9304.4140
C01221=-69.367,47.903,52.090,175.6152,2.4524,-9304.6279
C01222=-65.749,45.859,50.519,179.2918,0.3544,-9304.8952
C01223=-62.766,44.675,49.019,-171.7723,-2.6325,-9305.4421
C01224=-60.171,44.975,47.946,-148.9708,13.5769,-9306.7764
C01225=-57.387,47.412,47.522,-150.4313,29.9610,-9309.5628
C01226=-54.990,50.108,47.503,-151.2787,31.2909,-9312.3404
C01227=-52.606,52.606,47.516,-149.9534,30.0465,-9315.0000
C01228=-50.108,54.990,47.503,-148.7091,28.7214,-9317.6596
C01229=-47.412,57.387,47.522,-150.0405,29.5697,-9320.4372
C01230=-44.975,60.171,47.946,-166.4223,31.0293,-9323.2236
C01231=-44.675,62.766,49.019,177.3675,8.2277,-9324.5579
C01232=-45.859,65.749,50.519,-179.6456,-0.7082,-9325.1048
C01233=-47.903,69.367,52.090,-177.5476,-4.3848,-9325.3721
C01234=-50.285,73.401,53.317,-176.5147,-6.5160,-9325.5860
C01235=-52.213,77.409,53.931,-178.1887,-7.2383,-9326.0000
C01236=-52.061,81.773,54.258,178.7124,-4.2314,-9327.5170
C01237=-49.741,85.881,54.525,178.4742,-1.7165,-9329.9212
C01238=-45.636,88.910,54.796,179.8779,-0.0649,-9332.8293
C01239=-40.787,91.296,54.976,179.9844,-0.0071,-9335.9270
C01240=-35.715,93.397,54.976,179.9840,-0.0060,-9339.0732
C01241=-30.600,95.138,54.796,179.8678,-0.0404,-9342.1702
C01242=-25.555,95.900,54.525,177.7079,0.1349,-9345.0788
C01243=-21.009,94.635,54.258,176.0979,2.0860,-9347.4833
C01244=-17.816,91.657,53.931,176.1414,6.4001,-9349.0002
C01245=-16.346,87.459,53.317,177.8411,7.0591,-9349.4136
C01246=-15.177,82.922,52.090,178.6288,4.8303,-9349.6281
C01247=-14.064,78.919,50.519,179.7498,0.7514,-9349.8955
C01248=-12.792,75.972,49.019,-176.0111,-7.6747,-9350.4423
C01249=-10.745,74.349,47.946,-149.1991,-14.2834,-9351.7765
C01250=-7.053,74.105,47.522,-141.0348,0.3657,-9354.5632
C01251=-3.453,74.315,47.503,-140.7427,2.4222,-9357.3397
C01252=0.000,74.396,47.516,-140.7158,0.0000,-9360.0000
C01253=0.000,73.003,49.219,-140.7316,-0.0001,-9360.0000
C01254=3.325,72.927,49.205,-140.7578,-2.3938,-9362.6105
C01255=6.839,72.729,49.225,-141.0811,-0.0240,-9365.3720
C01256=10.483,73.017,49.677,-150.1638,14.9630,-9368.1701
C01257=12.469,74.753,50.822,-176.8894,6.5490,-9369.4699
C01258=13.691,77.880,52.422,179.5579,-1.4288,-9369.9705
C01259=14.768,82.123,54.099,178.6140,-5.2247,-9370.1944
C01260=15.905,86.934,55.407,177.9156,-7.3526,-9370.3679
C01261=17.335,91.395,56.062,176.2006,-6.7488,-9370.7398
C01262=20.556,94.581,56.410,175.9685,-2.2822,-9372.2618
C01263=25.196,95.965,56.695,177.6326,-0.1678,-9374.7112
C01264=30.373,95.213,56.983,179.8606,0.0424,-9377.6927
C01265=35.638,93.426,57.174,179.9832,0.0063,-9380.8797
C01266=40.862,91.262,57.174,179.9837,0.0074,-9384.1202
C01267=45.849,88.802,56.983,179.8715,0.0686,-9387.3076
C01268=50.042,85.674,56.695,178.4441,1.7930,-9390.2891
C01269=52.343,81.414,56.410,178.7594,4.4610,-9392.7379
C01270=52.368,76.884,56.062,-177.8971,7.4427,-9394.2600
C01271=50.225,72.718,55.407,-176.2521,6.6721,-9394.6321
C01272=47.627,68.512,54.099,-177.2776,4.6745,-9394.8056
C01273=45.389,64.750,52.422,-179.3021,1.3229,-9395.0300
C01274=44.041,61.675,50.822,177.5521,-6.8204,-9395.5299
C01275=44.219,59.044,49.677,-167.7797,-30.7331,-9396.8301
C01276=46.591,56.263,49.225,-150.2631,-29.7114,-9399.6279
C01277=49.216,53.919,49.205,-148.7368,-28.7232,-9402.3891
C01278=51.621,51.621,49.219,-149.9674,-30.0326,-9405.0000
C01279=53.919,49.216,49.205,-151.2767,-31.2632,-9407.6109
C01280=56.263,46.591,49.225,-150.2876,-29.7354,-9410.3721
C01281=59.044,44.219,49.677,-149.2668,-12.2210,-9413.1699
C01282=61.675,44.041,50.822,-173.1796,2.4479,-9414.4701
C01283=64.750,45.389,52.422,178.6771,-0.6979,-9414.9700
C01284=68.512,47.627,54.099,175.3255,-2.7224,-9415.1944
C01285=72.718,50.225,55.407,173.3279,-3.7479,-9415.3679
C01286=76.884,52.368,56.062,172.5573,-2.1029,-9415.7400
C01287=81.414,52.343,56.410,175.5390,1.2406,-9417.2621
C01288=85.674,50.042,56.695,178.2070,1.5559,-9419.7109
C01289=88.802,45.849,56.983,179.9314,0.1285,-9422.6924
C01290=91.262,40.862,57.174,179.9926,0.0163,-9425.8798
C01291=93.426,35.638,57.174,179.9937,0.0168,-9429.1203
C01292=95.213,30.373,56.983,179.9576,0.1394,-9432.3073
C01293=95.965,25.196,56.695,-179.8322,2.3674,-9435.2888
C01294=94.581,20.556,56.410,-177.7178,4.0315,-9437.7382
C01295=91.395,17.335,56.062,-173.2512,3.7994,-9439.2602
C01296=86.934,15.905,55.407,-172.6474,2.0844,-9439.6321
C01297=82.123,14.768,54.099,-174.7753,1.3860,-9439.8056
C01298=77.880,13.691,52.422,-178.5712,0.4421,-9440.0295
C01299=74.753,12.469,50.822,173.4510,-3.1106,-9440.5301
C01300=73.017,10.483,49.677,165.0370,-29.8362,-9441.8299
C01301=72.729,6.839,49.225,-179.9760,-38.9189,-9444.6280
C01302=72.927,3.325,49.205,-177.6062,-39.2422,-9447.3895
C01303=73.003,0.000,49.219,-179.9999,-39.2684,-9450.0000
C01304=72.927,-3.325,49.205,177.6063,-39.2423,-9452.6105
C01305=72.729,-6.839,49.225,179.9785,-38.9186,-9455.3720
C01306=73.017,-10.483,49.677,-165.0374,-29.8367,-9458.1701
C01307=74.753,-12.469,50.822,-173.4510,-3.1106,-9459.4699
C01308=77.880,-13.691,52.422,178.5712,0.4421,-9459.9705
C01309=82.123,-14.768,54.099,174.7753,1.3860,-9460.1944
C01310=86.934,-15.905,55.407,172.6474,2.0844,-9460.3679
C01311=91.395,-17.335,56.062,173.2512,3.7994,-9460.7398
C01312=94.581,-20.556,56.410,177.7178,4.0315,-9462.2618
C01313=95.965,-25.196,56.695,179.8322,2.3674,-9464.7112
C01314=95.213,-30.373,56.983,-179.9576,0.1394,-9467.6927
C01315=93.426,-35.638,57.174,-179.9937,0.0168,-9470.8797
C01316=91.262,-40.862,57.174,-179.9926,0.0163,-9474.1202
C01317=88.802,-45.849,56.983,-179.9314,0.1285,-9477.3076
C01318=85.674,-50.042,56.695,-178.2070,1.5559,-9480.2891
C01319=81.414,-52.343,56.410,-175.5390,1.2406,-9482.7379
C01320=76.884,-52.368,56.062,-172.5573,-2.1029,-9484.2600
C01321=72.718,-50.225,55.407,-173.3279,-3.7479,-9484.6321
C01322=68.512,-47.627,54.099,-175.3255,-2.7224,-9484.8056
C01323=64.750,-45.389,52.422,-178.6771,-0.6979,-9485.0300
C01324=61.675,-44.041,50.822,173.1796,2.4479,-9485.5299
C01325=59.044,-44.219,49.677,149.2669,-12.2203,-9486.8301
C01326=56.263,-46.591,49.225,150.2886,-29.7369,-9489.6279
C01327=53.919,-49.216,49.205,151.2768,-31.2632,-9492.3891
C01328=51.621,-51.621,49.219,149.9674,-30.0326,-9495.0000
C01329=49.216,-53.919,49.205,148.7368,-28.7233,-9497.6109
C01330=46.591,-56.263,49.225,150.2646,-29.7124,-9500.3721
C01331=44.219,-59.044,49.677,167.7790,-30.7332,-9503.1699
C01332=44.041,-61.675,50.822,-177.5521,-6.8204,-9504.4701
C01333=45.389,-64.750,52.422,179.3021,1.3229,-9504.9700
C01334=47.627,-68.512,54.099,177.2776,4.6745,-9505.1944
C01335=50.225,-72.718,55.407,176.2521,6.6721,-9505.3679
C01336=52.368,-76.884,56.062,177.8971,7.4427,-9505.7400
C01337=52.343,-81.414,56.410,-178.7594,4.4610,-9507.2621
C01338=50.042,-85.674,56.695,-178.4441,1.7930,-9509.7109
C01339=45.849,-88.802,56.983,-179.8715,0.0686,-9512.6924
C01340=40.862,-91.262,57.174,-179.9837,0.0074,-9515.8798
C01341=35.638,-93.426,57.174,-179.9832,0.0063,-9519.1203
C01342=30.373,-95.213,56.983,-179.8606,0.0424,-9522.3073
C01343=25.196,-95.965,56.695,-177.6326,-0.1678,-9525.2888
C01344=20.556,-94.581,56.410,-175.9685,-2.2822,-9527.7382
C01345=17.335,-91.395,56.062,-176.2006,-6.7488,-9529.2602
C01346=15.905,-86.934,55.407,-177.9156,-7.3526,-9529.6321
C01347=14.768,-82.123,54.099,-178.6140,-5.2247,-9529.8056
C01348=13.691,-77.880,52.422,-179.5579,-1.4288,-9530.0295
C01349=12.469,-74.753,50.822,176.8894,6.5490,-9530.5301
C01350=10.483,-73.017,49.677,150.1638,14.9630,-9531.8299
C01351=6.839,-72.729,49.225,141.0811,-0.0240,-9534.6280
C01352=3.325,-72.927,49.205,140.7578,-2.3938,-9537.3895
C01353=0.000,-73.003,49.219,140.7316,-0.0001,-9540.0000
C01354=0.000,-73.003,49.219,140.7316,-0.0001,-9540.0000
C01355=-3.325,-72.927,49.205,140.7577,2.3937,-9542.6105
C01356=-6.839,-72.729,49.225,141.0814,0.0215,-9545.3720
C01357=-10.483,-73.017,49.677,150.1633,-14.9626,-9548.1701
C01358=-12.469,-74.753,50.822,176.8894,-6.5490,-9549.4699
C01359=-13.691,-77.880,52.422,-179.5579,1.4288,-9549.9705
C01360=-14.768,-82.123,54.099,-178.6140,5.2247,-9550.1944
C01361=-15.905,-86.934,55.407,-177.9156,7.3526,-9550.3679
C01362=-17.335,-91.395,56.062,-176.2006,6.7488,-9550.7398
C01363=-20.556,-94.581,56.410,-175.9685,2.2822,-9552.2618
C01364=-25.196,-95.965,56.695,-177.6326,0.1678,-9554.7112
C01365=-30.373,-95.213,56.983,-179.8606,-0.0424,-9557.6927
C01366=-35.638,-93.426,57.174,-179.9832,-0.0063,-9560.8797
C01367=-40.862,-91.262,57.174,-179.9837,-0.0074,-9564.1202
C01368=-45.849,-88.802,56.983,-179.8715,-0.0686,-9567.3076
C01369=-50.042,-85.674,56.695,-178.4441,-1.7930,-9570.2891
C01370=-52.343,-81.414,56.410,-178.7594,-4.4610,-9572.7379
C01371=-52.368,-76.884,56.062,177.8971,-7.4427,-9574.2600
C01372=-50.225,-72.718,55.407,176.2521,-6.6721,-9574.6321
C01373=-47.627,-68.512,54.099,177.2776,-4.6745,-9574.8056
C01374=-45.389,-64.750,52.422,179.3021,-1.3229,-9575.0300
C01375=-44.041,-61.675,50.822,-177.5521,6.8204,-9575.5299
C01376=-44.219,-59.044,49.677,167.7797,30.7331,-9576.8301
C01377=-46.591,-56.263,49.225,150.2631,29.7114,-9579.6279
C01378=-49.216,-53.919,49.205,148.7368,28.7232,-9582.3891
C01379=-51.621,-51.621,49.219,149.9674,30.0326,-9585.0000
C01380=-53.919,-49.216,49.205,151.2767,31.2632,-9587.6109
C01381=-56.263,-46.591,49.225,150.2876,29.7354,-9590.3721
C01382=-59.044,-44.219,49.677,149.2668,12.2210,-9593.1699
C01383=-61.675,-44.041,50.822,173.1796,-2.4479,-9594.4701
C01384=-64.750,-45.389,52.422,-178.6771,0.6979,-9594.9700
C01385=-68.512,-47.627,54.099,-175.3255,2.7224,-9595.1944
C01386=-72.718,-50.225,55.407,-173.3279,3.7479,-9595.3679
C01387=-76.884,-52.368,56.062,-172.5573,2.1029,-9595.7400
C01388=-81.414,-52.343,56.410,-175.5390,-1.2406,-9597.2621
C01389=-85.674,-50.042,56.695,-178.2070,-1.5559,-9599.7109
C01390=-88.802,-45.849,56.983,-179.9314,-0.1285,-9602.6924
C01391=-91.262,-40.862,57.174,-179.9926,-0.0163,-9605.8798
C01392=-93.426,-35.638,57.174,-179.9937,-0.0168,-9609.1203
C01393=-95.213,-30.373,56.983,-179.9576,-0.1394,-9612.3073
C01394=-95.965,-25.196,56.695,179.8322,-2.3674,-9615.2888
C01395=-94.581,-20.556,56.410,177.7178,-4.0315,-9617.7382
C01396=-91.395,-17.335,56.062,173.2512,-3.7994,-9619.2602
C01397=-86.934,-15.905,55.407,172.6474,-2.0844,-9619.6321
C01398=-82.123,-14.768,54.099,174.7753,-1.3860,-9619.8056
C01399=-77.880,-13.691,52.422,178.5712,-0.4421,-9620.0295
C01400=-74.753,-12.469,50.822,-173.4510,3.1106,-9620.5301
C01401=-73.017,-10.483,49.677,-165.0370,29.8362,-9621.8299
C01402=-72.729,-6.839,49.225,179.9760,38.9189,-9624.6280
C01403=-72.927,-3.325,49.205,177.6062,39.2422,-9627.3895
C01404=-73.003,0.000,49.219,179.9999,39.2684,-9630.0000
C01405=-72.927,3.325,49.205,-177.6063,39.2423,-9632.6105
C01406=-72.729,6.839,49.225,-179.9785,38.9186,-9635.3720
C01407=-73.017,10.483,49.677,165.0374,29.8367,-9638.1701
C01408=-74.753,12.469,50.822,173.4510,3.1106,-9639.4699
C01409=-77.880,13.691,52.422,-178.5712,-0.4421,-9639.9705
C01410=-82.123,14.768,54.099,-174.7753,-1.3860,-9640.1944
C01411=-86.934,15.905,55.407,-172.6474,-2.0844,-9640.3679
C01412=-91.395,17.335,56.062,-173.2512,-3.7994,-9640.7398
C01413=-94.581,20.556,56.410,-177.7178,-4.0315,-9642.2618
C01414=-95.965,25.196,56.695,-179.8322,-2.3674,-9644.7112
C01415=-95.213,30.373,56.983,179.9576,-0.1394,-9647.6927
C01416=-93.426,35.638,57.174,179.9937,-0.0168,-9650.8797
C01417=-91.262,40.862,57.174,179.9926,-0.0163,-9654.1202
C01418=-88.802,45.849,56.983,179.9314,-0.1285,-9657.3076
C01419=-85.674,50.042,56.695,178.2070,-1.5559,-9660.2891
C01420=-81.414,52.343,56.410,175.5390,-1.2406,-9662.7379
C01421=-76.884,52.368,56.062,172.5573,2.1029,-9664.2600
C01422=-72.718,50.225,55.407,173.3279,3.7479,-9664.6321
C01423=-68.512,47.627,54.099,175.3255,2.7224,-9664.8056
C01424=-64.750,45.389,52.422,178.6771,0.6979,-9665.0300
C01425=-61.675,44.041,50.822,-173.1796,-2.4479,-9665.5299
C01426=-59.044,44.219,49.677,-149.2669,12.2203,-9666.8301
C01427=-56.263,46.591,49.225,-150.2886,29.7369,-9669.6279
C01428=-53.919,49.216,49.205,-151.2768,31.2632,-9672.3891
C01429=-51.621,51.621,49.219,-149.9674,30.0326,-9675.0000
C01430=-49.216,53.919,49.205,-148.7368,28.7233,-9677.6109
C01431=-46.591,56.263,49.225,-150.2646,29.7124,-9680.3721
C01432=-44.219,59.044,49.677,-167.7790,30.7332,-9683.1699
C01433=-44.041,61.675,50.822,177.5521,6.8204,-9684.4701
C01434=-45.389,64.750,52.422,-179.3021,-1.3229,-9684.9700
C01435=-47.627,68.512,54.099,-177.2776,-4.6745,-9685.1944
C01436=-50.225,72.718,55.407,-176.2521,-6.6721,-9685.3679
C01437=-52.368,76.884,56.062,-177.8971,-7.4427,-9685.7400
C01438=-52.343,81.414,56.410,178.7594,-4.4610,-9687.2621
C01439=-50.042,85.674,56.695,178.4441,-1.7930,-9689.7109
C01440=-45.849,88.802,56.983,179.8715,-0.0686,-9692.6924
C01441=-40.862,91.262,57.174,179.9837,-0.0074,-9695.8798
C01442=-35.638,93.426,57.174,179.9832,-0.0063,-9699.1203
C01443=-30.373,95.213,56.983,179.8606,-0.0424,-9702.3073
C01444=-25.196,95.965,56.695,177.6326,0.1678,-9705.2888
C01445=-20.556,94.581,56.410,175.9685,2.2822,-9707.7382
C01446=-17.335,91.395,56.062,176.2006,6.7488,-9709.2602
C01447=-15.905,86.934,55.407,177.9156,7.3526,-9709.6321
C01448=-14.768,82.123,54.099,178.6140,5.2247,-9709.8056
C01449=-13.691,77.880,52.422,179.5579,1.4288,-9710.0295
C01450=-12.469,74.753,50.822,-176.8894,-6.5490,-9710.5301
C01451=-10.483,73.017,49.677,-150.1633,-14.9626,-9711.8299
C01452=-6.839,72.729,49.225,-141.0814,0.0215,-9714.6280
C01453=-3.325,72.927,49.205,-140.7577,2.3937,-9717.3895
C01454=0.000,73.003,49.219,-140.7316,-0.0001,-9720.0000
C01455=0.000,71.612,50.923,-140.8208,-0.0002,-9720.0000
C01456=3.198,71.541,50.909,-140.8461,-2.3571,-9722.5595
C01457=6.625,71.354,50.929,-141.2051,0.3291,-9725.3045
C01458=10.220,71.688,51.410,-151.2344,15.5138,-9728.1135
C01459=12.146,73.537,52.627,-177.6255,5.4535,-9729.3788
C01460=13.319,76.847,54.328,179.4145,-2.0293,-9729.8327
C01461=14.363,81.331,56.111,178.6204,-5.5448,-9730.0151
C01462=15.469,86.415,57.500,178.0046,-7.5648,-9730.1489
C01463=16.861,91.137,58.195,176.2963,-7.0136,-9730.4816
C01464=20.110,94.527,58.564,175.8846,-2.4532,-9732.0102
C01465=24.842,96.029,58.865,177.5784,-0.1990,-9734.5040
C01466=30.149,95.287,59.171,179.8550,0.0439,-9737.5575
C01467=35.562,93.456,59.373,179.9827,0.0065,-9740.8329
C01468=40.937,91.230,59.373,179.9831,0.0077,-9744.1669
C01469=46.059,88.697,59.171,179.8665,0.0715,-9747.4422
C01470=50.337,85.469,58.865,178.4278,1.8534,-9750.4960
C01471=52.621,81.060,58.564,178.8209,4.6406,-9752.9901
C01472=52.521,76.366,58.195,-177.6396,7.5626,-9754.5184
C01473=50.167,72.043,57.500,-176.0374,6.7604,-9754.8513
C01474=47.354,67.666,56.111,-177.0453,4.8968,-9754.9851
C01475=44.921,63.757,54.328,-178.9786,1.8489,-9755.1672
C01476=43.410,60.587,52.627,177.8131,-5.5306,-9755.6212
C01477=43.464,57.918,51.410,-169.1369,-30.3048,-9756.8860
C01478=45.770,55.140,50.929,-150.5612,-29.7906,-9759.6950
C01479=48.325,52.849,50.909,-148.8319,-28.6632,-9762.4397
C01480=50.637,50.637,50.923,-150.0461,-29.9537,-9765.0000
C01481=52.848,48.326,50.909,-151.3368,-31.1682,-9767.5591
C01482=55.140,45.770,50.930,-150.2084,-29.4371,-9770.3050
C01483=57.918,43.464,51.410,-149.6951,-10.8637,-9773.1140
C01484=60.587,43.410,52.627,-174.4694,2.1869,-9774.3788
C01485=63.757,44.921,54.328,178.1511,-1.0214,-9774.8328
C01486=67.666,47.354,56.111,175.1032,-2.9547,-9775.0149
C01487=72.043,50.167,57.500,173.2396,-3.9626,-9775.1487
C01488=76.366,52.521,58.195,172.4374,-2.3604,-9775.4816
C01489=81.060,52.621,58.564,175.3594,1.1791,-9777.0099
C01490=85.469,50.337,58.865,178.1466,1.5722,-9779.5040
C01491=88.697,46.059,59.171,179.9285,0.1335,-9782.5578
C01492=91.230,40.937,59.373,179.9923,0.0169,-9785.8331
C01493=93.456,35.562,59.373,179.9935,0.0173,-9789.1671
C01494=95.287,30.149,59.171,179.9561,0.1450,-9792.4425
C01495=96.029,24.842,58.865,-179.8010,2.4216,-9795.4960
C01496=94.527,20.110,58.564,-177.5468,4.1154,-9797.9898
C01497=91.137,16.861,58.195,-172.9864,3.7037,-9799.5184
C01498=86.415,15.469,57.500,-172.4352,1.9954,-9799.8511
C01499=81.331,14.363,56.111,-174.4552,1.3796,-9799.9849
C01500=76.847,13.319,54.328,-177.9707,0.5855,-9800.1673
C01501=73.537,12.146,52.627,174.5465,-2.3745,-9800.6212
C01502=71.688,10.220,51.410,164.4862,-28.7656,-9801.8865
C01503=71.354,6.625,50.929,179.6709,-38.7949,-9804.6955
C01504=71.541,3.198,50.909,-177.6429,-39.1539,-9807.4405
C01505=71.612,0.000,50.923,-179.9998,-39.1792,-9810.0000
C01506=71.541,-3.198,50.909,177.6428,-39.1539,-9812.5595
C01507=71.354,-6.626,50.930,-179.6684,-38.7945,-9815.3053
C01508=71.688,-10.221,51.410,-164.4865,-28.7660,-9818.1143
C01509=73.537,-12.146,52.627,-174.5465,-2.3745,-9819.3788
C01510=76.847,-13.319,54.328,177.9707,0.5855,-9819.8327
C01511=81.331,-14.363,56.111,174.4552,1.3796,-9820.0151
C01512=86.415,-15.469,57.500,172.4352,1.9954,-9820.1489
C01513=91.137,-16.861,58.195,172.9864,3.7037,-9820.4816
C01514=94.527,-20.110,58.564,177.5468,4.1154,-9822.0102
C01515=96.029,-24.842,58.865,179.8010,2.4216,-9824.5040
C01516=95.287,-30.149,59.171,-179.9561,0.1450,-9827.5575
C01517=93.456,-35.562,59.373,-179.9935,0.0173,-9830.8329
C01518=91.230,-40.937,59.373,-179.9923,0.0169,-9834.1669
C01519=88.697,-46.059,59.171,-179.9285,0.1335,-9837.4422
C01520=85.469,-50.337,58.865,-178.1466,1.5722,-9840.4960
C01521=81.060,-52.621,58.564,-175.3594,1.1791,-9842.9901
C01522=76.366,-52.521,58.195,-172.4374,-2.3604,-9844.5184
C01523=72.043,-50.167,57.500,-173.2396,-3.9626,-9844.8513
C01524=67.666,-47.354,56.111,-175.1032,-2.9547,-9844.9851
C01525=63.757,-44.921,54.328,-178.1511,-1.0214,-9845.1672
C01526=60.587,-43.410,52.627,174.4694,2.1869,-9845.6212
C01527=57.918,-43.464,51.410,149.6952,-10.8631,-9846.8860
C01528=55.140,-45.770,50.929,150.2094,-29.4388,-9849.6950
C01529=52.849,-48.325,50.909,151.3368,-31.1681,-9852.4397
C01530=50.637,-50.637,50.923,150.0463,-29.9539,-9855.0000
C01531=48.326,-52.848,50.909,148.8318,-28.6632,-9857.5591
C01532=45.770,-55.140,50.930,150.5629,-29.7916,-9860.3050
C01533=43.464,-57.918,51.410,169.1363,-30.3049,-9863.1140
C01534=43.410,-60.587,52.627,-177.8131,-5.5306,-9864.3788
C01535=44.921,-63.757,54.328,178.9786,1.8489,-9864.8328
C01536=47.354,-67.666,56.111,177.0453,4.8968,-9865.0149
C01537=50.167,-72.043,57.500,176.0374,6.7604,-9865.1487
C01538=52.521,-76.366,58.195,177.6396,7.5626,-9865.4816
C01539=52.621,-81.060,58.564,-178.8209,4.6406,-9867.0099
C01540=50.337,-85.469,58.865,-178.4278,1.8534,-9869.5040
C01541=46.059,-88.697,59.171,-179.8665,0.0715,-9872.5578
C01542=40.937,-91.230,59.373,-179.9831,0.0077,-9875.8331
C01543=35.562,-93.456,59.373,-179.9827,0.0065,-9879.1671
C01544=30.149,-95.287,59.171,-179.8550,0.0439,-9882.4425
C01545=24.842,-96.029,58.865,-177.5784,-0.1990,-9885.4960
C01546=20.110,-94.527,58.564,-175.8846,-2.4532,-9887.9898
C01547=16.861,-91.137,58.195,-176.2963,-7.0136,-9889.5184
C01548=15.469,-86.415,57.500,-178.0046,-7.5648,-9889.8511
C01549=14.363,-81.331,56.111,-178.6204,-5.5448,-9889.9849
C01550=13.319,-76.847,54.328,-179.4145,-2.0293,-9890.1673
C01551=12.146,-73.537,52.627,177.6255,5.4535,-9890.6212
C01552=10.220,-71.688,51.410,151.2344,15.5138,-9891.8865
C01553=6.625,-71.354,50.929,141.2051,0.3291,-9894.6955
C01554=3.198,-71.541,50.909,140.8461,-2.3571,-9897.4405
C01555=0.000,-71.612,50.923,140.8208,-0.0002,-9900.0000
C01556=0.000,-71.612,50.923,140.8208,-0.0002,-9900.0000
C01557=-3.198,-71.541,50.909,140.8461,2.3572,-9902.5595
C01558=-6.626,-71.354,50.930,141.2055,-0.3316,-9905.3053
C01559=-10.221,-71.688,51.410,151.2340,-15.5135,-9908.1143
C01560=-12.146,-73.537,52.627,177.6255,-5.4535,-9909.3788
C01561=-13.319,-76.847,54.328,-179.4145,2.0293,-9909.8327
C01562=-14.363,-81.331,56.111,-178.6204,5.5448,-9910.0151
C01563=-15.469,-86.415,57.500,-178.0046,7.5648,-9910.1489
C01564=-16.861,-91.137,58.195,-176.2963,7.0136,-9910.4816
C01565=-20.110,-94.527,58.564,-175.8846,2.4532,-9912.0102
C01566=-24.842,-96.029,58.865,-177.5784,0.1990,-9914.5040
C01567=-30.149,-95.287,59.171,-179.8550,-0.0439,-9917.5575
C01568=-35.562,-93.456,59.373,-179.9827,-0.0065,-9920.8329
C01569=-40.937,-91.230,59.373,-179.9831,-0.0077,-9924.1669
C01570=-46.059,-88.697,59.171,-179.8665,-0.0715,-9927.4422
C01571=-50.337,-85.469,58.865,-178.4278,-1.8534,-9930.4960
C01572=-52.621,-81.060,58.564,-178.8209,-4.6406,-9932.9901
C01573=-52.521,-76.366,58.195,177.6396,-7.5626,-9934.5184
C01574=-50.167,-72.043,57.500,176.0374,-6.7604,-9934.8513
C01575=-47.354,-67.666,56.111,177.0453,-4.8968,-9934.9851
C01576=-44.921,-63.757,54.328,178.9786,-1.8489,-9935.1672
C01577=-43.410,-60.587,52.627,-177.8131,5.5306,-9935.6212
C01578=-43.464,-57.918,51.410,169.1369,30.3048,-9936.8860
C01579=-45.770,-55.140,50.929,150.5612,29.7906,-9939.6950
C01580=-48.325,-52.849,50.909,148.8319,28.6632,-9942.4397
C01581=-50.637,-50.637,50.923,150.0461,29.9537,-9945.0000
C01582=-52.848,-48.326,50.909,151.3368,31.1682,-9947.5591
C01583=-55.140,-45.770,50.930,150.2084,29.4371,-9950.3050
C01584=-57.918,-43.464,51.410,149.6951,10.8637,-9953.1140
C01585=-60.587,-43.410,52.627,174.4694,-2.1869,-9954.3788
C01586=-63.757,-44.921,54.328,-178.1511,1.0214,-9954.8328
C01587=-67.666,-47.354,56.111,-175.1032,2.9547,-9955.0149
C01588=-72.043,-50.167,57.500,-173.2396,3.9626,-9955.1487
C01589=-76.366,-52.521,58.195,-172.4374,2.3604,-9955.4816
C01590=-81.060,-52.621,58.564,-175.3594,-1.1791,-9957.0099
C01591=-85.469,-50.337,58.865,-178.1466,-1.5722,-9959.5040
C01592=-88.697,-46.059,59.171,-179.9285,-0.1335,-9962.5578
C01593=-91.230,-40.937,59.373,-179.9923,-0.0169,-9965.8331
C01594=-93.456,-35.562,59.373,-179.9935,-0.0173,-9969.1671
C01595=-95.287,-30.149,59.171,-179.9561,-0.1450,-9972.4425
C01596=-96.029,-24.842,58.865,179.8010,-2.4216,-9975.4960
C01597=-94.527,-20.110,58.564,177.5468,-4.1154,-9977.9898
C01598=-91.137,-16.861,58.195,172.9864,-3.7037,-9979.5184
C01599=-86.415,-15.469,57.500,172.4352,-1.9954,-9979.8511
C01600=-81.331,-14.363,56.111,174.4552,-1.3796,-9979.9849
C01601=-76.847,-13.319,54.328,177.9707,-0.5855,-9980.1673
C01602=-73.537,-12.146,52.627,-174.5465,2.3745,-9980.6212
C01603=-71.688,-10.220,51.410,-164.4862,28.7656,-9981.8865
C01604=-71.354,-6.625,50.929,-179.6709,38.7949,-9984.6955
C01605=-71.541,-3.198,50.909,177.6429,39.1539,-9987.4405
C01606=-71.612,0.000,50.923,179.9998,39.1792,-9990.0000
C01607=-71.541,3.198,50.909,-177.6428,39.1539,-9992.5595
C01608=-71.354,6.626,50.930,179.6684,38.7945,-9995.3053
C01609=-71.688,10.221,51.410,164.4865,28.7660,-9998.1143
C01610=-73.537,12.146,52.627,174.5465,2.3745,-9999.3788
C01611=-76.847,13.319,54.328,-177.9707,-0.5855,-9999.8327
C01612=-81.331,14.363,56.111,-174.4552,-1.3796,-10000.0151
C01613=-86.415,15.469,57.500,-172.4352,-1.9954,-10000.1489
C01614=-91.137,16.861,58.195,-172.9864,-3.7037,-10000.4816
C01615=-94.527,20.110,58.564,-177.5468,-4.1154,-10002.0102
C01616=-96.029,24.842,58.865,-179.8010,-2.4216,-10004.5040
C01617=-95.287,30.149,59.171,179.9561,-0.1450,-10007.5575
C01618=-93.456,35.562,59.373,179.9935,-0.0173,-10010.8329
C01619=-91.230,40.937,59.373,179.9923,-0.0169,-10014.1669
C01620=-88.697,46.059,59.171,179.9285,-0.1335,-10017.4422
C01621=-85.469,50.337,58.865,178.1466,-1.5722,-10020.4960
C01622=-81.060,52.621,58.564,175.3594,-1.1791,-10022.9901
C01623=-76.366,52.521,58.195,172.4374,2.3604,-10024.5184
C01624=-72.043,50.167,57.500,173.2396,3.9626,-10024.8513
C01625=-67.666,47.354,56.111,175.1032,2.9547,-10024.9851
C01626=-63.757,44.921,54.328,178.1511,1.0214,-10025.1672
C01627=-60.587,43.410,52.627,-174.4694,-2.1869,-10025.6212
C01628=-57.918,43.464,51.410,-149.6952,10.8631,-10026.8860
C01629=-55.140,45.770,50.929,-150.2094,29.4388,-10029.6950
C01630=-52.849,48.325,50.909,-151.3368,31.1681,-10032.4397
C01631=-50.637,50.637,50.923,-150.0463,29.9539,-10035.0000
C01632=-48.326,52.848,50.909,-148.8318,28.6632,-10037.5591
C01633=-45.770,55.140,50.930,-150.5629,29.7916,-10040.3050
C01634=-43.464,57.918,51.410,-169.1363,30.3049,-10043.1140
C01635=-43.410,60.587,52.627,177.8131,5.5306,-10044.3788
C01636=-44.921,63.757,54.328,-178.9786,-1.8489,-10044.8328
C01637=-47.354,67.666,56.111,-177.0453,-4.8968,-10045.0149
C01638=-50.167,72.043,57.500,-176.0374,-6.7604,-10045.1487
C01639=-52.521,76.366,58.195,-177.6396,-7.5626,-10045.4816
C01640=-52.621,81.060,58.564,178.8209,-4.6406,-10047.0099
C01641=-50.337,85.469,58.865,178.4278,-1.8534,-10049.5040
C01642=-46.059,88.697,59.171,179.8665,-0.0715,-10052.5578
C01643=-40.937,91.230,59.373,179.9831,-0.0077,-10055.8331
C01644=-35.562,93.456,59.373,179.9827,-0.0065,-10059.1671
C01645=-30.149,95.287,59.171,179.8550,-0.0439,-10062.4425
C01646=-24.842,96.029,58.865,177.5784,0.1990,-10065.4960
C01647=-20.110,94.527,58.564,175.8846,2.4532,-10067.9898
C01648=-16.861,91.137,58.195,176.2963,7.0136,-10069.5184
C01649=-15.469,86.415,57.500,178.0046,7.5648,-10069.8511
C01650=-14.363,81.331,56.111,178.6204,5.5448,-10069.9849
C01651=-13.319,76.847,54.328,179.4145,2.0293,-10070.1673
C01652=-12.146,73.537,52.627,-177.6255,-5.4535,-10070.6212
C01653=-10.221,71.688,51.410,-151.2340,-15.5135,-10071.8857
C01654=-6.626,71.354,50.930,-141.2055,-0.3316,-10074.6947
C01655=-3.198,71.541,50.909,-140.8461,2.3572,-10077.4405
C01656=0.000,71.612,50.923,-140.8208,-0.0002,-10080.0000
C01657=0.000,70.224,52.630,-140.9842,-0.0003,-10080.0000
C01658=3.072,70.158,52.615,-141.0087,-2.3123,-10082.5072
C01659=6.412,69.984,52.637,-141.4077,0.6880,-10085.2349
C01660=9.959,70.362,53.146,-152.3999,15.9321,-10088.0561
C01661=11.825,72.328,54.436,-178.2362,4.4065,-10089.2852
C01662=12.951,75.822,56.240,179.3107,-2.5537,-10089.6930
C01663=13.963,80.549,58.128,178.6435,-5.7936,-10089.8344
C01664=15.041,85.905,59.597,178.1039,-7.6987,-10089.9312
C01665=16.396,90.884,60.330,176.4208,-7.1953,-10090.2265
C01666=19.672,94.474,60.719,175.8447,-2.5954,-10091.7624
C01667=24.496,96.092,61.037,177.5461,-0.2275,-10094.3014
C01668=29.931,95.359,61.359,179.8510,0.0449,-10097.4259
C01669=35.488,93.484,61.571,179.9823,0.0066,-10100.7876
C01670=41.009,91.197,61.571,179.9828,0.0078,-10104.2123
C01671=46.265,88.593,61.359,179.8629,0.0736,-10107.5744
C01672=50.626,85.269,61.037,178.4250,1.8965,-10110.6985
C01673=52.893,80.714,60.719,178.8932,4.7688,-10113.2374
C01674=52.671,75.858,60.330,-177.4212,7.6040,-10114.7737
C01675=50.109,71.379,59.597,-175.8716,6.7862,-10115.0694
C01676=47.084,66.830,58.128,-176.8518,5.0569,-10115.1660
C01677=44.457,62.772,56.240,-178.6807,2.2931,-10115.3073
C01678=42.782,59.505,54.436,178.1262,-4.3612,-10115.7148
C01679=42.712,56.796,53.146,-170.4736,-29.7489,-10116.9441
C01680=44.952,54.020,52.637,-150.9334,-29.8046,-10119.7651
C01681=47.437,51.781,52.615,-148.9950,-28.5406,-10122.4931
C01682=49.656,49.656,52.630,-150.1903,-29.8094,-10125.0000
C01683=51.781,47.437,52.615,-151.4594,-31.0052,-10127.5069
C01684=54.020,44.952,52.637,-150.1944,-29.0648,-10130.2349
C01685=56.796,42.711,53.146,-150.2510,-9.5269,-10133.0566
C01686=59.505,42.782,54.436,-175.6388,1.8738,-10134.2852
C01687=62.772,44.457,56.240,177.7069,-1.3193,-10134.6927
C01688=66.830,47.084,58.128,174.9431,-3.1482,-10134.8340
C01689=71.379,50.109,59.597,173.2138,-4.1284,-10134.9306
C01690=75.858,52.671,60.330,172.3960,-2.5788,-10135.2263
C01691=80.714,52.893,60.719,175.2312,1.1068,-10136.7626
C01692=85.269,50.626,61.037,178.1035,1.5750,-10139.3015
C01693=88.593,46.265,61.359,179.9264,0.1371,-10142.4256
C01694=91.197,41.009,61.571,179.9922,0.0172,-10145.7877
C01695=93.484,35.488,61.571,179.9934,0.0177,-10149.2124
C01696=95.359,29.931,61.359,179.9551,0.1490,-10152.5741
C01697=96.092,24.496,61.037,-179.7725,2.4539,-10155.6986
C01698=94.474,19.672,60.719,-177.4046,4.1553,-10158.2376
C01699=90.884,16.396,60.330,-172.8047,3.5792,-10159.7735
C01700=85.905,15.041,59.597,-172.3013,1.8961,-10160.0688
C01701=80.549,13.963,58.128,-174.2064,1.3565,-10160.1656
C01702=75.822,12.951,56.240,-177.4463,0.6893,-10160.3070
C01703=72.328,11.825,54.436,175.5935,-1.7638,-10160.7148
C01704=70.362,9.959,53.146,164.0679,-27.6001,-10161.9439
C01705=69.984,6.412,52.637,179.3120,-38.5923,-10164.7651
C01706=70.158,3.072,52.615,-177.6877,-38.9913,-10167.4928
C01707=70.224,0.000,52.630,-179.9997,-39.0158,-10170.0000
C01708=70.158,-3.071,52.615,177.6875,-38.9914,-10172.5064
C01709=69.984,-6.412,52.637,-179.3094,-38.5919,-10175.2349
C01710=70.362,-9.959,53.146,-164.0682,-27.6005,-10178.0561
C01711=72.328,-11.825,54.436,-175.5935,-1.7638,-10179.2852
C01712=75.822,-12.951,56.240,177.4463,0.6893,-10179.6930
C01713=80.549,-13.963,58.128,174.2064,1.3565,-10179.8344
C01714=85.905,-15.041,59.597,172.3013,1.8961,-10179.9312
C01715=90.884,-16.396,60.330,172.8047,3.5792,-10180.2265
C01716=94.474,-19.672,60.719,177.4046,4.1553,-10181.7624
C01717=96.092,-24.496,61.037,179.7725,2.4539,-10184.3014
C01718=95.359,-29.931,61.359,-179.9551,0.1490,-10187.4259
C01719=93.484,-35.488,61.571,-179.9934,0.0177,-10190.7876
C01720=91.197,-41.009,61.571,-179.9922,0.0172,-10194.2123
C01721=88.593,-46.265,61.359,-179.9264,0.1371,-10197.5744
C01722=85.269,-50.626,61.037,-178.1035,1.5750,-10200.6985
C01723=80.714,-52.893,60.719,-175.2312,1.1068,-10203.2374
C01724=75.858,-52.671,60.330,-172.3960,-2.5788,-10204.7737
C01725=71.379,-50.109,59.597,-173.2138,-4.1284,-10205.0694
C01726=66.830,-47.084,58.128,-174.9431,-3.1482,-10205.1660
C01727=62.772,-44.457,56.240,-177.7069,-1.3193,-10205.3073
C01728=59.505,-42.782,54.436,175.6388,1.8738,-10205.7148
C01729=56.796,-42.712,53.146,150.2511,-9.5264,-10206.9441
C01730=54.020,-44.952,52.637,150.1954,-29.0666,-10209.7651
C01731=51.781,-47.437,52.615,151.4594,-31.0050,-10212.4931
C01732=49.656,-49.656,52.630,150.1906,-29.8097,-10215.0000
C01733=47.437,-51.781,52.615,148.9948,-28.5406,-10217.5069
C01734=44.952,-54.020,52.637,150.9352,-29.8056,-10220.2349
C01735=42.711,-56.796,53.146,170.4731,-29.7490,-10223.0566
C01736=42.782,-59.505,54.436,-178.1262,-4.3612,-10224.2852
C01737=44.457,-62.772,56.240,178.6807,2.2931,-10224.6927
C01738=47.084,-66.830,58.128,176.8518,5.0569,-10224.8340
C01739=50.109,-71.379,59.597,175.8716,6.7862,-10224.9306
C01740=52.671,-75.858,60.330,177.4212,7.6040,-10225.2263
C01741=52.893,-80.714,60.719,-178.8932,4.7688,-10226.7626
